LIN {X 0,Y 187.079,Z 92.881,A -85,B 0,C 180,E1 -22258.507,E2 -22258.507} C_VEL
LIN {X 0,Y 185.729,Z 90.066,A -85,B 0,C 180,E1 -22258.924,E2 -22258.924} C_VEL
LIN {X 0,Y 185.6,Z 89.366,A -85,B 0,C 180,E1 -22259.069,E2 -22259.069} C_VEL
LIN {X 0,Y 185.536,Z 89.372,A -85,B 0,C 180,E1 -22263.556,E2 -22263.556} C_VEL
LIN {X 0,Y 185.545,Z 89.369,A -85,B 0,C 180,E1 -22267.304,E2 -22267.304} C_VEL
LIN {X 0,Y 185.487,Z 89.376,A -85,B 0,C 180,E1 -22270.731,E2 -22270.731} C_VEL
LIN {X 0,Y 185.461,Z 89.378,A -85,B 0,C 180,E1 -22276.055,E2 -22276.055} C_VEL
LIN {X 0,Y 185.469,Z 89.375,A -85,B 0,C 180,E1 -22279.896,E2 -22279.896} C_VEL
LIN {X 0,Y 185.508,Z 89.375,A -85,B 0,C 180,E1 -22282.712,E2 -22282.712} C_VEL
LIN {X 0,Y 185.548,Z 89.369,A -85,B 0,C 180,E1 -22287.976,E2 -22287.976} C_VEL
LIN {X 0,Y 185.584,Z 89.362,A -85,B 0,C 180,E1 -22290.576,E2 -22290.576} C_VEL
LIN {X 0,Y 185.59,Z 89.361,A -85,B 0,C 180,E1 -22295.383,E2 -22295.383} C_VEL
LIN {X 0,Y 185.61,Z 89.358,A -85,B 0,C 180,E1 -22300.076,E2 -22300.076} C_VEL
LIN {X 0,Y 185.698,Z 89.324,A -85,B 0,C 180,E1 -22304.638,E2 -22304.638} C_VEL
LIN {X 0,Y 185.891,Z 89.329,A -85,B 0,C 180,E1 -22309.418,E2 -22309.418} C_VEL
LIN {X 0,Y 185.949,Z 89.301,A -85,B 0,C 180,E1 -22313.49,E2 -22313.49} C_VEL
LIN {X 0,Y 186.208,Z 89.273,A -85,B 0,C 180,E1 -22317.837,E2 -22317.837} C_VEL
LIN {X 0,Y 186.41,Z 89.262,A -85,B 0,C 180,E1 -22320,E2 -22320} C_VEL
LIN {X 0,Y 185.915,Z 89.319,A -85,B 0,C 180,E1 -22324.336,E2 -22324.336} C_VEL
LIN {X 0,Y 185.982,Z 89.316,A -85,B 0,C 180,E1 -22328.694,E2 -22328.694} C_VEL
LIN {X 0,Y 185.726,Z 89.351,A -85,B 0,C 180,E1 -22333.123,E2 -22333.123} C_VEL
LIN {X 0,Y 185.689,Z 89.356,A -85,B 0,C 180,E1 -22337.625,E2 -22337.625} C_VEL
LIN {X 0,Y 185.578,Z 89.369,A -85,B 0,C 180,E1 -22342.254,E2 -22342.254} C_VEL
LIN {X 0,Y 185.513,Z 89.381,A -85,B 0,C 180,E1 -22347.04,E2 -22347.04} C_VEL
LIN {X 0,Y 185.546,Z 89.375,A -85,B 0,C 180,E1 -22349.499,E2 -22349.499} C_VEL
LIN {X 0,Y 185.501,Z 89.381,A -85,B 0,C 180,E1 -22354.632,E2 -22354.632} C_VEL
LIN {X 0,Y 185.508,Z 89.378,A -85,B 0,C 180,E1 -22357.313,E2 -22357.313} C_VEL
LIN {X 0,Y 185.474,Z 89.382,A -85,B 0,C 180,E1 -22360.725,E2 -22360.725} C_VEL
LIN {X 0,Y 185.463,Z 89.382,A -85,B 0,C 180,E1 -22366.054,E2 -22366.054} C_VEL
LIN {X 0,Y 185.447,Z 89.388,A -85,B 0,C 180,E1 -22366.815,E2 -22366.815} C_VEL
LIN {X 0,Y 187.546,Z 97.212,A -85,B 0,C 180,E1 -22371.041,E2 -22371.041} C_VEL
LIN {X 0,Y 194.525,Z 112.749,A -85,B 0,C 180,E1 -22373.096,E2 -22373.096} C_VEL
LIN {X 0,Y 199.839,Z 126.939,A -85,B 0,C 180,E1 -22374.634,E2 -22374.634} C_VEL
LIN {X 0,Y 202.047,Z 149.722,A -85,B 0,C 180,E1 -22375.924,E2 -22375.924} C_VEL
LIN {X 0,Y 203.001,Z 161.188,A -85,B 0,C 180,E1 -22376.533,E2 -22376.533} C_VEL
LIN {X 0,Y 201.967,Z 186.96,A -85,B 0,C 180,E1 -22377.398,E2 -22377.398} C_VEL
LIN {X 0,Y 201.164,Z 192.812,A -85,B 0,C 180,E1 -22377.503,E2 -22377.503} C_VEL
LIN {X 0,Y 195.507,Z 209.786,A -85,B 0,C 180,E1 -22377.456,E2 -22377.456} C_VEL
LIN {X 0,Y 194.095,Z 215.48,A -85,B 0,C 180,E1 -22377.666,E2 -22377.666} C_VEL
LIN {X 0,Y 193.836,Z 217.383,A -85,B 0,C 180,E1 -22377.795,E2 -22377.795} C_VEL
LIN {X 0,Y 192.139,Z 229.824,A -85,B 0,C 180,E1 -22378.891,E2 -22378.891} C_VEL
LIN {X 0,Y 189.978,Z 241.772,A -85,B 0,C 180,E1 -22380.344,E2 -22380.344} C_VEL
LIN {X 0,Y 187.729,Z 252.645,A -85,B 0,C 180,E1 -22382.097,E2 -22382.097} C_VEL
LIN {X 0,Y 185.608,Z 261.462,A -85,B 0,C 180,E1 -22383.884,E2 -22383.884} C_VEL
LIN {X 0,Y 183.397,Z 270.914,A -85,B 0,C 180,E1 -22386.273,E2 -22386.273} C_VEL
LIN {X 0,Y 181.019,Z 279.181,A -85,B 0,C 180,E1 -22388.842,E2 -22388.842} C_VEL
LIN {X 0,Y 179.368,Z 286.6,A -85,B 0,C 180,E1 -22391.732,E2 -22391.732} C_VEL
LIN {X 0,Y 177.815,Z 293.562,A -85,B 0,C 180,E1 -22395.113,E2 -22395.113} C_VEL
LIN {X 0,Y 176.781,Z 299.125,A -85,B 0,C 180,E1 -22398.534,E2 -22398.534} C_VEL
LIN {X 0,Y 176.302,Z 303.475,A -85,B 0,C 180,E1 -22401.98,E2 -22401.98} C_VEL
LIN {X 0,Y 176.263,Z 306.729,A -85,B 0,C 180,E1 -22405.426,E2 -22405.426} C_VEL
LIN {X 0,Y 176.338,Z 308.334,A -85,B 0,C 180,E1 -22407.716,E2 -22407.716} C_VEL
LIN {X 0,Y 176.495,Z 309.519,A -85,B 0,C 180,E1 -22410,E2 -22410} C_VEL
LIN {X 0,Y 176.316,Z 310.226,A -85,B 0,C 180,E1 -22412.284,E2 -22412.284} C_VEL
LIN {X 0,Y 176.232,Z 310.534,A -85,B 0,C 180,E1 -22414.575,E2 -22414.575} C_VEL
LIN {X 0,Y 176.383,Z 309.99,A -85,B 0,C 180,E1 -22419.171,E2 -22419.171} C_VEL
LIN {X 0,Y 176.861,Z 309.117,A -85,B 0,C 180,E1 -22421.46,E2 -22421.46} C_VEL
LIN {X 0,Y 178.546,Z 306.157,A -85,B 0,C 180,E1 -22425.994,E2 -22425.994} C_VEL
LIN {X 0,Y 180.7,Z 302.835,A -85,B 0,C 180,E1 -22429.305,E2 -22429.305} C_VEL
LIN {X 0,Y 183.398,Z 298.468,A -85,B 0,C 180,E1 -22432.533,E2 -22432.533} C_VEL
LIN {X 0,Y 187.098,Z 291.917,A -85,B 0,C 180,E1 -22436.191,E2 -22436.191} C_VEL
LIN {X 0,Y 191.062,Z 284.767,A -85,B 0,C 180,E1 -22439.169,E2 -22439.169} C_VEL
LIN {X 0,Y 195.634,Z 275.903,A -85,B 0,C 180,E1 -22441.998,E2 -22441.998} C_VEL
LIN {X 0,Y 200.264,Z 265.844,A -85,B 0,C 180,E1 -22444.464,E2 -22444.464} C_VEL
LIN {X 0,Y 204.349,Z 255.58,A -85,B 0,C 180,E1 -22446.389,E2 -22446.389} C_VEL
LIN {X 0,Y 208.228,Z 244.222,A -85,B 0,C 180,E1 -22448.022,E2 -22448.022} C_VEL
LIN {X 0,Y 211.569,Z 232.42,A -85,B 0,C 180,E1 -22449.289,E2 -22449.289} C_VEL
LIN {X 0,Y 214.263,Z 219.437,A -85,B 0,C 180,E1 -22450.3,E2 -22450.3} C_VEL
LIN {X 0,Y 216.25,Z 205.853,A -85,B 0,C 180,E1 -22450.98,E2 -22450.98} C_VEL
LIN {X 0,Y 218.563,Z 169.214,A -85,B 0,C 180,E1 -22452.133,E2 -22452.133} C_VEL
LIN {X 0,Y 217.377,Z 159.103,A -85,B 0,C 180,E1 -22452.939,E2 -22452.939} C_VEL
LIN {X 0,Y 211.594,Z 145.25,A -85,B 0,C 180,E1 -22455.352,E2 -22455.352} C_VEL
LIN {X 0,Y 206.029,Z 134.045,A -85,B 0,C 180,E1 -22457.813,E2 -22457.813} C_VEL
LIN {X 0,Y 201.532,Z 125.851,A -85,B 0,C 180,E1 -22459.965,E2 -22459.965} C_VEL
LIN {X 0,Y 196.559,Z 117.494,A -85,B 0,C 180,E1 -22462.566,E2 -22462.566} C_VEL
LIN {X 0,Y 192.905,Z 111.765,A -85,B 0,C 180,E1 -22464.664,E2 -22464.664} C_VEL
LIN {X 0,Y 188.825,Z 105.716,A -85,B 0,C 180,E1 -22467.254,E2 -22467.254} C_VEL
LIN {X 0,Y 185.057,Z 100.378,A -85,B 0,C 180,E1 -22469.954,E2 -22469.954} C_VEL
LIN {X 0,Y 183.131,Z 97.941,A -85,B 0,C 180,E1 -22471.462,E2 -22471.462} C_VEL
LIN {X 0,Y 180.355,Z 94.307,A -85,B 0,C 180,E1 -22473.883,E2 -22473.883} C_VEL
LIN {X 0,Y 179.145,Z 92.283,A -85,B 0,C 180,E1 -22475.199,E2 -22475.199} C_VEL
LIN {X 0,Y 178.547,Z 90.23,A -85,B 0,C 180,E1 -22478.041,E2 -22478.041} C_VEL
LIN {X 0,Y 178.673,Z 90.218,A -85,B 0,C 180,E1 -22481.658,E2 -22481.658} C_VEL
LIN {X 0,Y 178.661,Z 90.221,A -85,B 0,C 180,E1 -22486.348,E2 -22486.348} C_VEL
LIN {X 0,Y 178.914,Z 90.196,A -85,B 0,C 180,E1 -22490.96,E2 -22490.96} C_VEL
LIN {X 0,Y 179.154,Z 90.152,A -85,B 0,C 180,E1 -22497.752,E2 -22497.752} C_VEL
LIN {X 0,Y 179.372,Z 90.132,A -85,B 0,C 180,E1 -22500,E2 -22500} C_VEL
LIN {X 0,Y 178.866,Z 90.189,A -85,B 0,C 180,E1 -22504.507,E2 -22504.507} C_VEL
LIN {X 0,Y 178.912,Z 90.181,A -85,B 0,C 180,E1 -22509.04,E2 -22509.04} C_VEL
LIN {X 0,Y 178.652,Z 90.367,A -85,B 0,C 180,E1 -22515.034,E2 -22515.034} C_VEL
LIN {X 0,Y 179.507,Z 92.842,A -85,B 0,C 180,E1 -22516.052,E2 -22516.052} C_VEL
LIN {X 0,Y 181.383,Z 94.994,A -85,B 0,C 180,E1 -22517.766,E2 -22517.766} C_VEL
LIN {X 0,Y 183.423,Z 96.333,A -85,B 0,C 180,E1 -22519.371,E2 -22519.371} C_VEL
LIN {X 0,Y 185.032,Z 99.289,A -85,B 0,C 180,E1 -22520.714,E2 -22520.714} C_VEL
LIN {X 0,Y 187.677,Z 101.543,A -85,B 0,C 180,E1 -22522.533,E2 -22522.533} C_VEL
LIN {X 0,Y 190.252,Z 105.409,A -85,B 0,C 180,E1 -22524.286,E2 -22524.286} C_VEL
LIN {X 0,Y 192.095,Z 107.229,A -85,B 0,C 180,E1 -22525.388,E2 -22525.388} C_VEL
LIN {X 0,Y 194.769,Z 110.861,A -85,B 0,C 180,E1 -22526.956,E2 -22526.956} C_VEL
LIN {X 0,Y 196.441,Z 113.104,A -85,B 0,C 180,E1 -22527.876,E2 -22527.876} C_VEL
LIN {X 0,Y 199.512,Z 117.279,A -85,B 0,C 180,E1 -22529.476,E2 -22529.476} C_VEL
LIN {X 0,Y 204.379,Z 124.152,A -85,B 0,C 180,E1 -22531.81,E2 -22531.81} C_VEL
LIN {X 0,Y 211.211,Z 134.963,A -85,B 0,C 180,E1 -22534.777,E2 -22534.777} C_VEL
LIN {X 0,Y 217.553,Z 146.272,A -85,B 0,C 180,E1 -22537.28,E2 -22537.28} C_VEL
LIN {X 0,Y 219.698,Z 150.374,A -85,B 0,C 180,E1 -22538.082,E2 -22538.082} C_VEL
LIN {X 0,Y 217.14,Z 189.325,A -85,B 0,C 180,E1 -22539.281,E2 -22539.281} C_VEL
LIN {X 0,Y 215.488,Z 202.678,A -85,B 0,C 180,E1 -22540.031,E2 -22540.031} C_VEL
LIN {X 0,Y 213.455,Z 214.164,A -85,B 0,C 180,E1 -22540.995,E2 -22540.995} C_VEL
LIN {X 0,Y 210.553,Z 226.047,A -85,B 0,C 180,E1 -22542.313,E2 -22542.313} C_VEL
LIN {X 0,Y 207.233,Z 236.837,A -85,B 0,C 180,E1 -22543.89,E2 -22543.89} C_VEL
LIN {X 0,Y 203.257,Z 247.568,A -85,B 0,C 180,E1 -22545.904,E2 -22545.904} C_VEL
LIN {X 0,Y 199.599,Z 256.292,A -85,B 0,C 180,E1 -22548.01,E2 -22548.01} C_VEL
LIN {X 0,Y 195.695,Z 264.272,A -85,B 0,C 180,E1 -22550.397,E2 -22550.397} C_VEL
LIN {X 0,Y 191.556,Z 272,A -85,B 0,C 180,E1 -22553.402,E2 -22553.402} C_VEL
LIN {X 0,Y 187.26,Z 279.067,A -85,B 0,C 180,E1 -22557.03,E2 -22557.03} C_VEL
LIN {X 0,Y 184.152,Z 283.709,A -85,B 0,C 180,E1 -22560.255,E2 -22560.255} C_VEL
LIN {X 0,Y 182.382,Z 286.142,A -85,B 0,C 180,E1 -22562.457,E2 -22562.457} C_VEL
LIN {X 0,Y 180.863,Z 288.109,A -85,B 0,C 180,E1 -22564.695,E2 -22564.695} C_VEL
LIN {X 0,Y 179.569,Z 289.65,A -85,B 0,C 180,E1 -22566.959,E2 -22566.959} C_VEL
LIN {X 0,Y 178.48,Z 290.741,A -85,B 0,C 180,E1 -22569.244,E2 -22569.244} C_VEL
LIN {X 0,Y 177.61,Z 291.439,A -85,B 0,C 180,E1 -22571.746,E2 -22571.746} C_VEL
LIN {X 0,Y 176.514,Z 291.56,A -85,B 0,C 180,E1 -22576.179,E2 -22576.179} C_VEL
LIN {X 0,Y 176.263,Z 291.008,A -85,B 0,C 180,E1 -22578.5,E2 -22578.5} C_VEL
LIN {X 0,Y 176.402,Z 288.697,A -85,B 0,C 180,E1 -22583.136,E2 -22583.136} C_VEL
LIN {X 0,Y 176.854,Z 285.866,A -85,B 0,C 180,E1 -22586.583,E2 -22586.583} C_VEL
LIN {X 0,Y 177.509,Z 282.036,A -85,B 0,C 180,E1 -22590,E2 -22590} C_VEL
LIN {X 0,Y 178.57,Z 277.089,A -85,B 0,C 180,E1 -22593.385,E2 -22593.385} C_VEL
LIN {X 0,Y 180.129,Z 270.873,A -85,B 0,C 180,E1 -22596.722,E2 -22596.722} C_VEL
LIN {X 0,Y 182.228,Z 263.095,A -85,B 0,C 180,E1 -22599.995,E2 -22599.995} C_VEL
LIN {X 0,Y 184.684,Z 253.401,A -85,B 0,C 180,E1 -22603.199,E2 -22603.199} C_VEL
LIN {X 0,Y 187.279,Z 243.315,A -85,B 0,C 180,E1 -22605.788,E2 -22605.788} C_VEL
LIN {X 0,Y 189.62,Z 233.3,A -85,B 0,C 180,E1 -22607.805,E2 -22607.805} C_VEL
LIN {X 0,Y 191.652,Z 222.453,A -85,B 0,C 180,E1 -22609.55,E2 -22609.55} C_VEL
LIN {X 0,Y 193.437,Z 210.502,A -85,B 0,C 180,E1 -22611.026,E2 -22611.026} C_VEL
LIN {X 0,Y 194.843,Z 197.397,A -85,B 0,C 180,E1 -22612.186,E2 -22612.186} C_VEL
LIN {X 0,Y 195.736,Z 184.28,A -85,B 0,C 180,E1 -22612.914,E2 -22612.914} C_VEL
LIN {X 0,Y 198.224,Z 129.371,A -85,B 0,C 180,E1 -22614.791,E2 -22614.791} C_VEL
LIN {X 0,Y 194.633,Z 120.748,A -85,B 0,C 180,E1 -22615.793,E2 -22615.793} C_VEL
LIN {X 0,Y 187.561,Z 106.659,A -85,B 0,C 180,E1 -22617.78,E2 -22617.78} C_VEL
LIN {X 0,Y 181.804,Z 96.696,A -85,B 0,C 180,E1 -22619.473,E2 -22619.473} C_VEL
LIN {X 0,Y 180.363,Z 94.19,A -85,B 0,C 180,E1 -22619.92,E2 -22619.92} C_VEL
LIN {X 0,Y 178.803,Z 91.62,A -85,B 0,C 180,E1 -22620.409,E2 -22620.409} C_VEL
LIN {X 0,Y 178.493,Z 90.248,A -85,B 0,C 180,E1 -22620.599,E2 -22620.599} C_VEL
LIN {X 0,Y 178.496,Z 90.248,A -85,B 0,C 180,E1 -22624.225,E2 -22624.225} C_VEL
LIN {X 0,Y 178.42,Z 90.26,A -85,B 0,C 180,E1 -22629.069,E2 -22629.069} C_VEL
LIN {X 0,Y 178.405,Z 90.258,A -85,B 0,C 180,E1 -22632.044,E2 -22632.044} C_VEL
LIN {X 0,Y 178.395,Z 90.256,A -85,B 0,C 180,E1 -22635.164,E2 -22635.164} C_VEL
LIN {X 0,Y 178.404,Z 90.259,A -85,B 0,C 180,E1 -22638.46,E2 -22638.46} C_VEL
LIN {X 0,Y 178.425,Z 90.252,A -85,B 0,C 180,E1 -22643.784,E2 -22643.784} C_VEL
LIN {X 0,Y 178.489,Z 90.249,A -85,B 0,C 180,E1 -22646.547,E2 -22646.547} C_VEL
LIN {X 0,Y 178.525,Z 90.24,A -85,B 0,C 180,E1 -22650.007,E2 -22650.007} C_VEL
LIN {X 0,Y 178.537,Z 90.239,A -85,B 0,C 180,E1 -22654.876,E2 -22654.876} C_VEL
LIN {X 0,Y 178.626,Z 90.222,A -85,B 0,C 180,E1 -22660.784,E2 -22660.784} C_VEL
LIN {X 0,Y 178.662,Z 90.215,A -85,B 0,C 180,E1 -22666.348,E2 -22666.348} C_VEL
LIN {X 0,Y 178.914,Z 90.195,A -85,B 0,C 180,E1 -22670.96,E2 -22670.96} C_VEL
LIN {X 0,Y 179.154,Z 90.15,A -85,B 0,C 180,E1 -22677.752,E2 -22677.752} C_VEL
LIN {X 0,Y 179.373,Z 90.138,A -85,B 0,C 180,E1 -22680,E2 -22680} C_VEL
LIN {X 0,Y 178.862,Z 90.197,A -85,B 0,C 180,E1 -22684.508,E2 -22684.508} C_VEL
LIN {X 0,Y 178.911,Z 90.195,A -85,B 0,C 180,E1 -22689.041,E2 -22689.041} C_VEL
LIN {X 0,Y 178.655,Z 90.23,A -85,B 0,C 180,E1 -22693.653,E2 -22693.653} C_VEL
LIN {X 0,Y 178.624,Z 90.233,A -85,B 0,C 180,E1 -22699.214,E2 -22699.214} C_VEL
LIN {X 0,Y 178.518,Z 90.245,A -85,B 0,C 180,E1 -22705.111,E2 -22705.111} C_VEL
LIN {X 0,Y 178.463,Z 90.258,A -85,B 0,C 180,E1 -22710.794,E2 -22710.794} C_VEL
LIN {X 0,Y 178.486,Z 90.254,A -85,B 0,C 180,E1 -22714.218,E2 -22714.218} C_VEL
LIN {X 0,Y 178.398,Z 90.263,A -85,B 0,C 180,E1 -22719.074,E2 -22719.074} C_VEL
LIN {X 0,Y 178.401,Z 90.263,A -85,B 0,C 180,E1 -22722.045,E2 -22722.045} C_VEL
LIN {X 0,Y 178.418,Z 90.378,A -85,B 0,C 180,E1 -22725.76,E2 -22725.76} C_VEL
LIN {X 0,Y 180.164,Z 96.881,A -85,B 0,C 180,E1 -22729.415,E2 -22729.415} C_VEL
LIN {X 0,Y 186.535,Z 110.257,A -85,B 0,C 180,E1 -22731.427,E2 -22731.427} C_VEL
LIN {X 0,Y 192.601,Z 125.371,A -85,B 0,C 180,E1 -22733.283,E2 -22733.283} C_VEL
LIN {X 0,Y 193.865,Z 128.929,A -85,B 0,C 180,E1 -22733.668,E2 -22733.668} C_VEL
LIN {X 0,Y 195.93,Z 151.227,A -85,B 0,C 180,E1 -22734.975,E2 -22734.975} C_VEL
LIN {X 0,Y 196.76,Z 162.292,A -85,B 0,C 180,E1 -22735.576,E2 -22735.576} C_VEL
LIN {X 0,Y 194.789,Z 206.829,A -85,B 0,C 180,E1 -22737.161,E2 -22737.161} C_VEL
LIN {X 0,Y 193.836,Z 217.383,A -85,B 0,C 180,E1 -22737.795,E2 -22737.795} C_VEL
LIN {X 0,Y 193.089,Z 221.163,A -85,B 0,C 180,E1 -22738.044,E2 -22738.044} C_VEL
LIN {X 0,Y 190.241,Z 228.451,A -85,B 0,C 180,E1 -22738.439,E2 -22738.439} C_VEL
LIN {X 0,Y 184.998,Z 238.939,A -85,B 0,C 180,E1 -22739.182,E2 -22739.182} C_VEL
LIN {X 0,Y 183.098,Z 244.152,A -85,B 0,C 180,E1 -22739.822,E2 -22739.822} C_VEL
LIN {X 0,Y 182.711,Z 245.852,A -85,B 0,C 180,E1 -22740.091,E2 -22740.091} C_VEL
LIN {X 0,Y 180.095,Z 256.718,A -85,B 0,C 180,E1 -22742.076,E2 -22742.076} C_VEL
LIN {X 0,Y 177.533,Z 266.947,A -85,B 0,C 180,E1 -22744.5,E2 -22744.5} C_VEL
LIN {X 0,Y 175.322,Z 275.52,A -85,B 0,C 180,E1 -22747.058,E2 -22747.058} C_VEL
LIN {X 0,Y 173.589,Z 281.649,A -85,B 0,C 180,E1 -22749.252,E2 -22749.252} C_VEL
LIN {X 0,Y 171.721,Z 289.545,A -85,B 0,C 180,E1 -22752.739,E2 -22752.739} C_VEL
LIN {X 0,Y 170.071,Z 296.759,A -85,B 0,C 180,E1 -22756.863,E2 -22756.863} C_VEL
LIN {X 0,Y 169.361,Z 301.565,A -85,B 0,C 180,E1 -22760.445,E2 -22760.445} C_VEL
LIN {X 0,Y 169.124,Z 305.224,A -85,B 0,C 180,E1 -22764.037,E2 -22764.037} C_VEL
LIN {X 0,Y 169.255,Z 307.84,A -85,B 0,C 180,E1 -22767.62,E2 -22767.62} C_VEL
LIN {X 0,Y 169.429,Z 309.056,A -85,B 0,C 180,E1 -22770,E2 -22770} C_VEL
LIN {X 0,Y 169.153,Z 310.116,A -85,B 0,C 180,E1 -22774.316,E2 -22774.316} C_VEL
LIN {X 0,Y 169.086,Z 310.075,A -85,B 0,C 180,E1 -22777.163,E2 -22777.163} C_VEL
LIN {X 0,Y 169.857,Z 308.813,A -85,B 0,C 180,E1 -22781.939,E2 -22781.939} C_VEL
LIN {X 0,Y 171.721,Z 305.907,A -85,B 0,C 180,E1 -22786.648,E2 -22786.648} C_VEL
LIN {X 0,Y 173.969,Z 302.637,A -85,B 0,C 180,E1 -22790.083,E2 -22790.083} C_VEL
LIN {X 0,Y 176.824,Z 298.327,A -85,B 0,C 180,E1 -22793.419,E2 -22793.419} C_VEL
LIN {X 0,Y 180.722,Z 291.842,A -85,B 0,C 180,E1 -22797.19,E2 -22797.19} C_VEL
LIN {X 0,Y 184.879,Z 284.794,A -85,B 0,C 180,E1 -22800.244,E2 -22800.244} C_VEL
LIN {X 0,Y 189.648,Z 276.013,A -85,B 0,C 180,E1 -22803.135,E2 -22803.135} C_VEL
LIN {X 0,Y 194.47,Z 266.071,A -85,B 0,C 180,E1 -22805.644,E2 -22805.644} C_VEL
LIN {X 0,Y 198.691,Z 255.981,A -85,B 0,C 180,E1 -22807.601,E2 -22807.601} C_VEL
LIN {X 0,Y 202.702,Z 244.802,A -85,B 0,C 180,E1 -22809.254,E2 -22809.254} C_VEL
LIN {X 0,Y 206.425,Z 232.262,A -85,B 0,C 180,E1 -22810.627,E2 -22810.627} C_VEL
LIN {X 0,Y 209.214,Z 219.401,A -85,B 0,C 180,E1 -22811.644,E2 -22811.644} C_VEL
LIN {X 0,Y 211.219,Z 206.356,A -85,B 0,C 180,E1 -22812.311,E2 -22812.311} C_VEL
LIN {X 0,Y 213.641,Z 170.417,A -85,B 0,C 180,E1 -22813.466,E2 -22813.466} C_VEL
LIN {X 0,Y 212.726,Z 162.146,A -85,B 0,C 180,E1 -22814.147,E2 -22814.147} C_VEL
LIN {X 0,Y 207.357,Z 149.125,A -85,B 0,C 180,E1 -22816.53,E2 -22816.53} C_VEL
LIN {X 0,Y 202.042,Z 138.081,A -85,B 0,C 180,E1 -22819.045,E2 -22819.045} C_VEL
LIN {X 0,Y 196.613,Z 128.146,A -85,B 0,C 180,E1 -22821.85,E2 -22821.85} C_VEL
LIN {X 0,Y 193.113,Z 122.307,A -85,B 0,C 180,E1 -22823.825,E2 -22823.825} C_VEL
LIN {X 0,Y 190.334,Z 117.733,A -85,B 0,C 180,E1 -22825.529,E2 -22825.529} C_VEL
LIN {X 0,Y 186.434,Z 111.75,A -85,B 0,C 180,E1 -22828.146,E2 -22828.146} C_VEL
LIN {X 0,Y 182.795,Z 106.363,A -85,B 0,C 180,E1 -22830.911,E2 -22830.911} C_VEL
LIN {X 0,Y 177.729,Z 99.455,A -85,B 0,C 180,E1 -22835.51,E2 -22835.51} C_VEL
LIN {X 0,Y 175.025,Z 96.393,A -85,B 0,C 180,E1 -22838.505,E2 -22838.505} C_VEL
LIN {X 0,Y 172.883,Z 94.324,A -85,B 0,C 180,E1 -22841.329,E2 -22841.329} C_VEL
LIN {X 0,Y 171.786,Z 92.097,A -85,B 0,C 180,E1 -22843.282,E2 -22843.282} C_VEL
LIN {X 0,Y 171.586,Z 91.097,A -85,B 0,C 180,E1 -22843.873,E2 -22843.873} C_VEL
LIN {X 0,Y 171.85,Z 91.08,A -85,B 0,C 180,E1 -22850.585,E2 -22850.585} C_VEL
LIN {X 0,Y 171.818,Z 91.08,A -85,B 0,C 180,E1 -22855.307,E2 -22855.307} C_VEL
LIN {X 0,Y 172.335,Z 91.008,A -85,B 0,C 180,E1 -22860,E2 -22860} C_VEL
LIN {X 0,Y 171.814,Z 91.068,A -85,B 0,C 180,E1 -22864.692,E2 -22864.692} C_VEL
LIN {X 0,Y 171.885,Z 91.271,A -85,B 0,C 180,E1 -22867.488,E2 -22867.488} C_VEL
LIN {X 0,Y 172.525,Z 93.251,A -85,B 0,C 180,E1 -22868.787,E2 -22868.787} C_VEL
LIN {X 0,Y 174.365,Z 95.792,A -85,B 0,C 180,E1 -22871.475,E2 -22871.475} C_VEL
LIN {X 0,Y 176.872,Z 97.237,A -85,B 0,C 180,E1 -22874.232,E2 -22874.232} C_VEL
LIN {X 0,Y 178.186,Z 100.016,A -85,B 0,C 180,E1 -22875.733,E2 -22875.733} C_VEL
LIN {X 0,Y 180.534,Z 102.228,A -85,B 0,C 180,E1 -22877.852,E2 -22877.852} C_VEL
LIN {X 0,Y 181.461,Z 102.963,A -85,B 0,C 180,E1 -22878.611,E2 -22878.611} C_VEL
LIN {X 0,Y 183.559,Z 106.305,A -85,B 0,C 180,E1 -22880.376,E2 -22880.376} C_VEL
LIN {X 0,Y 185.749,Z 108.325,A -85,B 0,C 180,E1 -22881.939,E2 -22881.939} C_VEL
LIN {X 0,Y 188.215,Z 111.879,A -85,B 0,C 180,E1 -22883.666,E2 -22883.666} C_VEL
LIN {X 0,Y 189.886,Z 113.752,A -85,B 0,C 180,E1 -22884.72,E2 -22884.72} C_VEL
LIN {X 0,Y 193.951,Z 119.332,A -85,B 0,C 180,E1 -22887.151,E2 -22887.151} C_VEL
LIN {X 0,Y 197.722,Z 124.622,A -85,B 0,C 180,E1 -22889.185,E2 -22889.185} C_VEL
LIN {X 0,Y 202.306,Z 131.456,A -85,B 0,C 180,E1 -22891.451,E2 -22891.451} C_VEL
LIN {X 0,Y 208.135,Z 140.952,A -85,B 0,C 180,E1 -22894.077,E2 -22894.077} C_VEL
LIN {X 0,Y 214.692,Z 153.106,A -85,B 0,C 180,E1 -22896.776,E2 -22896.776} C_VEL
LIN {X 0,Y 212.202,Z 189.729,A -85,B 0,C 180,E1 -22897.925,E2 -22897.925} C_VEL
LIN {X 0,Y 210.489,Z 203.084,A -85,B 0,C 180,E1 -22898.685,E2 -22898.685} C_VEL
LIN {X 0,Y 208.186,Z 215.487,A -85,B 0,C 180,E1 -22899.749,E2 -22899.749} C_VEL
LIN {X 0,Y 205.125,Z 227.154,A -85,B 0,C 180,E1 -22901.082,E2 -22901.082} C_VEL
LIN {X 0,Y 201.318,Z 238.818,A -85,B 0,C 180,E1 -22902.852,E2 -22902.852} C_VEL
LIN {X 0,Y 197.645,Z 248.181,A -85,B 0,C 180,E1 -22904.669,E2 -22904.669} C_VEL
LIN {X 0,Y 193.421,Z 257.736,A -85,B 0,C 180,E1 -22907.056,E2 -22907.056} C_VEL
LIN {X 0,Y 188.602,Z 266.875,A -85,B 0,C 180,E1 -22909.999,E2 -22909.999} C_VEL
LIN {X 0,Y 184.186,Z 274.505,A -85,B 0,C 180,E1 -22913.254,E2 -22913.254} C_VEL
LIN {X 0,Y 180.008,Z 280.796,A -85,B 0,C 180,E1 -22916.866,E2 -22916.866} C_VEL
LIN {X 0,Y 176.893,Z 285.113,A -85,B 0,C 180,E1 -22920.223,E2 -22920.223} C_VEL
LIN {X 0,Y 174.312,Z 288.321,A -85,B 0,C 180,E1 -22923.672,E2 -22923.672} C_VEL
LIN {X 0,Y 172.887,Z 289.896,A -85,B 0,C 180,E1 -22926.014,E2 -22926.014} C_VEL
LIN {X 0,Y 171.728,Z 291.048,A -85,B 0,C 180,E1 -22928.388,E2 -22928.388} C_VEL
LIN {X 0,Y 170.593,Z 291.854,A -85,B 0,C 180,E1 -22931.359,E2 -22931.359} C_VEL
LIN {X 0,Y 169.531,Z 291.966,A -85,B 0,C 180,E1 -22935.598,E2 -22935.598} C_VEL
LIN {X 0,Y 169.214,Z 291.477,A -85,B 0,C 180,E1 -22938.015,E2 -22938.015} C_VEL
LIN {X 0,Y 169.268,Z 289.231,A -85,B 0,C 180,E1 -22942.845,E2 -22942.845} C_VEL
LIN {X 0,Y 169.739,Z 286.463,A -85,B 0,C 180,E1 -22946.439,E2 -22946.439} C_VEL
LIN {X 0,Y 170.381,Z 282.704,A -85,B 0,C 180,E1 -22950,E2 -22950} C_VEL
LIN {X 0,Y 171.506,Z 277.829,A -85,B 0,C 180,E1 -22953.524,E2 -22953.524} C_VEL
LIN {X 0,Y 173.096,Z 271.697,A -85,B 0,C 180,E1 -22956.997,E2 -22956.997} C_VEL
LIN {X 0,Y 175.284,Z 264.059,A -85,B 0,C 180,E1 -22960.395,E2 -22960.395} C_VEL
LIN {X 0,Y 177.813,Z 254.485,A -85,B 0,C 180,E1 -22963.719,E2 -22963.719} C_VEL
LIN {X 0,Y 180.472,Z 244.58,A -85,B 0,C 180,E1 -22966.4,E2 -22966.4} C_VEL
LIN {X 0,Y 182.918,Z 234.796,A -85,B 0,C 180,E1 -22968.481,E2 -22968.481} C_VEL
LIN {X 0,Y 185.049,Z 224.218,A -85,B 0,C 180,E1 -22970.277,E2 -22970.277} C_VEL
LIN {X 0,Y 187.057,Z 211.535,A -85,B 0,C 180,E1 -22971.924,E2 -22971.924} C_VEL
LIN {X 0,Y 188.529,Z 198.803,A -85,B 0,C 180,E1 -22973.116,E2 -22973.116} C_VEL
LIN {X 0,Y 189.452,Z 186.403,A -85,B 0,C 180,E1 -22973.865,E2 -22973.865} C_VEL
LIN {X 0,Y 192.002,Z 130.643,A -85,B 0,C 180,E1 -22975.851,E2 -22975.851} C_VEL
LIN {X 0,Y 185.329,Z 116.24,A -85,B 0,C 180,E1 -22977.801,E2 -22977.801} C_VEL
LIN {X 0,Y 178.679,Z 103.908,A -85,B 0,C 180,E1 -22979.836,E2 -22979.836} C_VEL
LIN {X 0,Y 174.98,Z 97.881,A -85,B 0,C 180,E1 -22981.018,E2 -22981.018} C_VEL
LIN {X 0,Y 173.262,Z 95.093,A -85,B 0,C 180,E1 -22981.59,E2 -22981.59} C_VEL
LIN {X 0,Y 171.822,Z 92.792,A -85,B 0,C 180,E1 -22982.08,E2 -22982.08} C_VEL
LIN {X 0,Y 171.394,Z 91.137,A -85,B 0,C 180,E1 -22982.296,E2 -22982.296} C_VEL
LIN {X 0,Y 171.407,Z 91.133,A -85,B 0,C 180,E1 -22985.032,E2 -22985.032} C_VEL
LIN {X 0,Y 171.381,Z 91.136,A -85,B 0,C 180,E1 -22988.817,E2 -22988.817} C_VEL
LIN {X 0,Y 171.323,Z 91.14,A -85,B 0,C 180,E1 -22994.217,E2 -22994.217} C_VEL
LIN {X 0,Y 171.336,Z 91.136,A -85,B 0,C 180,E1 -22998.982,E2 -22998.982} C_VEL
LIN {X 0,Y 171.389,Z 91.134,A -85,B 0,C 180,E1 -23002.042,E2 -23002.042} C_VEL
LIN {X 0,Y 171.4,Z 91.127,A -85,B 0,C 180,E1 -23005.093,E2 -23005.093} C_VEL
LIN {X 0,Y 171.452,Z 91.122,A -85,B 0,C 180,E1 -23010.535,E2 -23010.535} C_VEL
LIN {X 0,Y 171.461,Z 91.121,A -85,B 0,C 180,E1 -23015.802,E2 -23015.802} C_VEL
LIN {X 0,Y 171.582,Z 91.098,A -85,B 0,C 180,E1 -23020.872,E2 -23020.872} C_VEL
LIN {X 0,Y 171.579,Z 91.091,A -85,B 0,C 180,E1 -23025.773,E2 -23025.773} C_VEL
LIN {X 0,Y 171.851,Z 91.076,A -85,B 0,C 180,E1 -23030.585,E2 -23030.585} C_VEL
LIN {X 0,Y 171.814,Z 91.047,A -85,B 0,C 180,E1 -23035.308,E2 -23035.308} C_VEL
LIN {X 0,Y 172.336,Z 91.015,A -85,B 0,C 180,E1 -23040,E2 -23040} C_VEL
LIN {X 0,Y 171.811,Z 91.075,A -85,B 0,C 180,E1 -23044.693,E2 -23044.693} C_VEL
LIN {X 0,Y 171.849,Z 91.072,A -85,B 0,C 180,E1 -23049.415,E2 -23049.415} C_VEL
LIN {X 0,Y 171.572,Z 91.111,A -85,B 0,C 180,E1 -23054.228,E2 -23054.228} C_VEL
LIN {X 0,Y 171.543,Z 91.113,A -85,B 0,C 180,E1 -23059.558,E2 -23059.558} C_VEL
LIN {X 0,Y 171.447,Z 91.127,A -85,B 0,C 180,E1 -23065.599,E2 -23065.599} C_VEL
LIN {X 0,Y 171.42,Z 91.135,A -85,B 0,C 180,E1 -23070.573,E2 -23070.573} C_VEL
LIN {X 0,Y 171.395,Z 91.138,A -85,B 0,C 180,E1 -23075.035,E2 -23075.035} C_VEL
LIN {X 0,Y 171.36,Z 91.141,A -85,B 0,C 180,E1 -23078.808,E2 -23078.808} C_VEL
LIN {X 0,Y 171.367,Z 91.284,A -85,B 0,C 180,E1 -23084.552,E2 -23084.552} C_VEL
LIN {X 0,Y 172.713,Z 96.273,A -85,B 0,C 180,E1 -23087.579,E2 -23087.579} C_VEL
LIN {X 0,Y 174.962,Z 100.629,A -85,B 0,C 180,E1 -23088.365,E2 -23088.365} C_VEL
LIN {X 0,Y 180.087,Z 111.356,A -85,B 0,C 180,E1 -23090.095,E2 -23090.095} C_VEL
LIN {X 0,Y 184.61,Z 122.124,A -85,B 0,C 180,E1 -23091.573,E2 -23091.573} C_VEL
LIN {X 0,Y 187.983,Z 131.446,A -85,B 0,C 180,E1 -23092.672,E2 -23092.672} C_VEL
LIN {X 0,Y 190.642,Z 161.189,A -85,B 0,C 180,E1 -23094.474,E2 -23094.474} C_VEL
LIN {X 0,Y 188.658,Z 205.888,A -85,B 0,C 180,E1 -23096.108,E2 -23096.108} C_VEL
LIN {X 0,Y 187.324,Z 219.248,A -85,B 0,C 180,E1 -23096.962,E2 -23096.962} C_VEL
LIN {X 0,Y 185.495,Z 231.462,A -85,B 0,C 180,E1 -23098.125,E2 -23098.125} C_VEL
LIN {X 0,Y 183.146,Z 243.777,A -85,B 0,C 180,E1 -23099.757,E2 -23099.757} C_VEL
LIN {X 0,Y 182.711,Z 245.852,A -85,B 0,C 180,E1 -23100.091,E2 -23100.091} C_VEL
LIN {X 0,Y 181.391,Z 249.288,A -85,B 0,C 180,E1 -23100.586,E2 -23100.586} C_VEL
LIN {X 0,Y 177.453,Z 254.474,A -85,B 0,C 180,E1 -23101.19,E2 -23101.19} C_VEL
LIN {X 0,Y 173.45,Z 259.47,A -85,B 0,C 180,E1 -23101.917,E2 -23101.917} C_VEL
LIN {X 0,Y 172.05,Z 262.576,A -85,B 0,C 180,E1 -23102.601,E2 -23102.601} C_VEL
LIN {X 0,Y 169.87,Z 270.865,A -85,B 0,C 180,E1 -23104.908,E2 -23104.908} C_VEL
LIN {X 0,Y 167.246,Z 279.285,A -85,B 0,C 180,E1 -23107.778,E2 -23107.778} C_VEL
LIN {X 0,Y 165.479,Z 286.319,A -85,B 0,C 180,E1 -23110.783,E2 -23110.783} C_VEL
LIN {X 0,Y 163.791,Z 293.195,A -85,B 0,C 180,E1 -23114.444,E2 -23114.444} C_VEL
LIN {X 0,Y 162.511,Z 299.495,A -85,B 0,C 180,E1 -23118.778,E2 -23118.778} C_VEL
LIN {X 0,Y 162.082,Z 303.581,A -85,B 0,C 180,E1 -23122.525,E2 -23122.525} C_VEL
LIN {X 0,Y 162.103,Z 306.169,A -85,B 0,C 180,E1 -23125.691,E2 -23125.691} C_VEL
LIN {X 0,Y 162.34,Z 308.586,A -85,B 0,C 180,E1 -23130,E2 -23130} C_VEL
LIN {X 0,Y 162.079,Z 309.676,A -85,B 0,C 180,E1 -23134.195,E2 -23134.195} C_VEL
LIN {X 0,Y 162.01,Z 309.7,A -85,B 0,C 180,E1 -23137.478,E2 -23137.478} C_VEL
LIN {X 0,Y 162.868,Z 308.498,A -85,B 0,C 180,E1 -23142.46,E2 -23142.46} C_VEL
LIN {X 0,Y 163.693,Z 307.279,A -85,B 0,C 180,E1 -23144.928,E2 -23144.928} C_VEL
LIN {X 0,Y 166.458,Z 303.629,A -85,B 0,C 180,E1 -23149.741,E2 -23149.741} C_VEL
LIN {X 0,Y 169.272,Z 299.728,A -85,B 0,C 180,E1 -23153.23,E2 -23153.23} C_VEL
LIN {X 0,Y 172.561,Z 294.722,A -85,B 0,C 180,E1 -23156.616,E2 -23156.616} C_VEL
LIN {X 0,Y 176.518,Z 288.471,A -85,B 0,C 180,E1 -23159.847,E2 -23159.847} C_VEL
LIN {X 0,Y 181.201,Z 280.71,A -85,B 0,C 180,E1 -23162.888,E2 -23162.888} C_VEL
LIN {X 0,Y 186.453,Z 271.023,A -85,B 0,C 180,E1 -23165.75,E2 -23165.75} C_VEL
LIN {X 0,Y 191.131,Z 261.05,A -85,B 0,C 180,E1 -23168.018,E2 -23168.018} C_VEL
LIN {X 0,Y 195.255,Z 251.208,A -85,B 0,C 180,E1 -23169.71,E2 -23169.71} C_VEL
LIN {X 0,Y 198.928,Z 240.546,A -85,B 0,C 180,E1 -23171.148,E2 -23171.148} C_VEL
LIN {X 0,Y 202.491,Z 227.731,A -85,B 0,C 180,E1 -23172.426,E2 -23172.426} C_VEL
LIN {X 0,Y 205.105,Z 215.098,A -85,B 0,C 180,E1 -23173.312,E2 -23173.312} C_VEL
LIN {X 0,Y 206.853,Z 201.747,A -85,B 0,C 180,E1 -23173.906,E2 -23173.906} C_VEL
LIN {X 0,Y 208.847,Z 171.574,A -85,B 0,C 180,E1 -23174.864,E2 -23174.864} C_VEL
LIN {X 0,Y 208.211,Z 165.369,A -85,B 0,C 180,E1 -23175.388,E2 -23175.388} C_VEL
LIN {X 0,Y 203.058,Z 152.645,A -85,B 0,C 180,E1 -23177.832,E2 -23177.832} C_VEL
LIN {X 0,Y 198.139,Z 142.284,A -85,B 0,C 180,E1 -23180.322,E2 -23180.322} C_VEL
LIN {X 0,Y 193.338,Z 133.198,A -85,B 0,C 180,E1 -23182.976,E2 -23182.976} C_VEL
LIN {X 0,Y 189.796,Z 127.132,A -85,B 0,C 180,E1 -23185.115,E2 -23185.115} C_VEL
LIN {X 0,Y 187.532,Z 123.291,A -85,B 0,C 180,E1 -23186.604,E2 -23186.604} C_VEL
LIN {X 0,Y 184.091,Z 117.83,A -85,B 0,C 180,E1 -23189.056,E2 -23189.056} C_VEL
LIN {X 0,Y 179.828,Z 111.341,A -85,B 0,C 180,E1 -23192.546,E2 -23192.546} C_VEL
LIN {X 0,Y 176.763,Z 107.144,A -85,B 0,C 180,E1 -23195.474,E2 -23195.474} C_VEL
LIN {X 0,Y 175.368,Z 105.075,A -85,B 0,C 180,E1 -23197.011,E2 -23197.011} C_VEL
LIN {X 0,Y 173.518,Z 103.132,A -85,B 0,C 180,E1 -23199.201,E2 -23199.201} C_VEL
LIN {X 0,Y 171.394,Z 100.773,A -85,B 0,C 180,E1 -23202.243,E2 -23202.243} C_VEL
LIN {X 0,Y 170.374,Z 98.365,A -85,B 0,C 180,E1 -23204.293,E2 -23204.293} C_VEL
LIN {X 0,Y 169.698,Z 97.955,A -85,B 0,C 180,E1 -23205.612,E2 -23205.612} C_VEL
LIN {X 0,Y 167.533,Z 96.687,A -85,B 0,C 180,E1 -23212.77,E2 -23212.77} C_VEL
LIN {X 0,Y 167.921,Z 96.571,A -85,B 0,C 180,E1 -23220,E2 -23220} C_VEL
LIN {X 0,Y 170.58,Z 98.229,A -85,B 0,C 180,E1 -23226.802,E2 -23226.802} C_VEL
LIN {X 0,Y 171.871,Z 101.192,A -85,B 0,C 180,E1 -23229.265,E2 -23229.265} C_VEL
LIN {X 0,Y 174.263,Z 103.474,A -85,B 0,C 180,E1 -23232.445,E2 -23232.445} C_VEL
LIN {X 0,Y 175.296,Z 104.149,A -85,B 0,C 180,E1 -23233.586,E2 -23233.586} C_VEL
LIN {X 0,Y 176.887,Z 107.062,A -85,B 0,C 180,E1 -23235.409,E2 -23235.409} C_VEL
LIN {X 0,Y 179.658,Z 109.692,A -85,B 0,C 180,E1 -23237.942,E2 -23237.942} C_VEL
LIN {X 0,Y 181.935,Z 113.072,A -85,B 0,C 180,E1 -23239.902,E2 -23239.902} C_VEL
LIN {X 0,Y 183.695,Z 114.857,A -85,B 0,C 180,E1 -23241.221,E2 -23241.221} C_VEL
LIN {X 0,Y 186.471,Z 118.651,A -85,B 0,C 180,E1 -23243.216,E2 -23243.216} C_VEL
LIN {X 0,Y 187.694,Z 120.217,A -85,B 0,C 180,E1 -23244.029,E2 -23244.029} C_VEL
LIN {X 0,Y 191.422,Z 125.425,A -85,B 0,C 180,E1 -23246.36,E2 -23246.36} C_VEL
LIN {X 0,Y 196.258,Z 132.421,A -85,B 0,C 180,E1 -23249.056,E2 -23249.056} C_VEL
LIN {X 0,Y 202.388,Z 142.225,A -85,B 0,C 180,E1 -23252.11,E2 -23252.11} C_VEL
LIN {X 0,Y 208.309,Z 152.989,A -85,B 0,C 180,E1 -23254.777,E2 -23254.777} C_VEL
LIN {X 0,Y 209.855,Z 156.007,A -85,B 0,C 180,E1 -23255.435,E2 -23255.435} C_VEL
LIN {X 0,Y 207.331,Z 190.749,A -85,B 0,C 180,E1 -23256.536,E2 -23256.536} C_VEL
LIN {X 0,Y 205.483,Z 204.239,A -85,B 0,C 180,E1 -23257.324,E2 -23257.324} C_VEL
LIN {X 0,Y 203.077,Z 216.438,A -85,B 0,C 180,E1 -23258.401,E2 -23258.401} C_VEL
LIN {X 0,Y 199.933,Z 227.9,A -85,B 0,C 180,E1 -23259.741,E2 -23259.741} C_VEL
LIN {X 0,Y 195.962,Z 239.495,A -85,B 0,C 180,E1 -23261.525,E2 -23261.525} C_VEL
LIN {X 0,Y 191.605,Z 250.069,A -85,B 0,C 180,E1 -23263.655,E2 -23263.655} C_VEL
LIN {X 0,Y 187.289,Z 259.131,A -85,B 0,C 180,E1 -23266.035,E2 -23266.035} C_VEL
LIN {X 0,Y 182.3,Z 268.097,A -85,B 0,C 180,E1 -23269.051,E2 -23269.051} C_VEL
LIN {X 0,Y 178.066,Z 275.003,A -85,B 0,C 180,E1 -23272.127,E2 -23272.127} C_VEL
LIN {X 0,Y 173.96,Z 280.863,A -85,B 0,C 180,E1 -23275.556,E2 -23275.556} C_VEL
LIN {X 0,Y 170.615,Z 285.254,A -85,B 0,C 180,E1 -23279.009,E2 -23279.009} C_VEL
LIN {X 0,Y 167.83,Z 288.532,A -85,B 0,C 180,E1 -23282.572,E2 -23282.572} C_VEL
LIN {X 0,Y 166.259,Z 290.142,A -85,B 0,C 180,E1 -23284.994,E2 -23284.994} C_VEL
LIN {X 0,Y 164.997,Z 291.337,A -85,B 0,C 180,E1 -23287.459,E2 -23287.459} C_VEL
LIN {X 0,Y 163.651,Z 292.253,A -85,B 0,C 180,E1 -23290.872,E2 -23290.872} C_VEL
LIN {X 0,Y 162.54,Z 292.373,A -85,B 0,C 180,E1 -23294.964,E2 -23294.964} C_VEL
LIN {X 0,Y 162.164,Z 291.933,A -85,B 0,C 180,E1 -23297.485,E2 -23297.485} C_VEL
LIN {X 0,Y 162.033,Z 291.053,A -85,B 0,C 180,E1 -23300.009,E2 -23300.009} C_VEL
LIN {X 0,Y 162.433,Z 288.571,A -85,B 0,C 180,E1 -23304.349,E2 -23304.349} C_VEL
LIN {X 0,Y 162.965,Z 284.728,A -85,B 0,C 180,E1 -23308.765,E2 -23308.765} C_VEL
LIN {X 0,Y 164.018,Z 280.306,A -85,B 0,C 180,E1 -23312.456,E2 -23312.456} C_VEL
LIN {X 0,Y 165.427,Z 274.711,A -85,B 0,C 180,E1 -23316.097,E2 -23316.097} C_VEL
LIN {X 0,Y 167.53,Z 267.694,A -85,B 0,C 180,E1 -23319.66,E2 -23319.66} C_VEL
LIN {X 0,Y 170.002,Z 258.944,A -85,B 0,C 180,E1 -23323.143,E2 -23323.143} C_VEL
LIN {X 0,Y 172.841,Z 248.99,A -85,B 0,C 180,E1 -23326.234,E2 -23326.234} C_VEL
LIN {X 0,Y 175.635,Z 238.782,A -85,B 0,C 180,E1 -23328.67,E2 -23328.67} C_VEL
LIN {X 0,Y 178.17,Z 227.501,A -85,B 0,C 180,E1 -23330.794,E2 -23330.794} C_VEL
LIN {X 0,Y 180.241,Z 215.842,A -85,B 0,C 180,E1 -23332.496,E2 -23332.496} C_VEL
LIN {X 0,Y 181.943,Z 203.095,A -85,B 0,C 180,E1 -23333.853,E2 -23333.853} C_VEL
LIN {X 0,Y 183.165,Z 189.525,A -85,B 0,C 180,E1 -23334.814,E2 -23334.814} C_VEL
LIN {X 0,Y 185.949,Z 132.679,A -85,B 0,C 180,E1 -23336.926,E2 -23336.926} C_VEL
LIN {X 0,Y 178.931,Z 117.621,A -85,B 0,C 180,E1 -23339.114,E2 -23339.114} C_VEL
LIN {X 0,Y 171.415,Z 104.014,A -85,B 0,C 180,E1 -23341.6,E2 -23341.6} C_VEL
LIN {X 0,Y 166.936,Z 96.811,A -85,B 0,C 180,E1 -23343.183,E2 -23343.183} C_VEL
LIN {X 0,Y 164.825,Z 93.715,A -85,B 0,C 180,E1 -23343.953,E2 -23343.953} C_VEL
LIN {X 0,Y 164.385,Z 92.005,A -85,B 0,C 180,E1 -23344.225,E2 -23344.225} C_VEL
LIN {X 0,Y 164.301,Z 92.017,A -85,B 0,C 180,E1 -23349.914,E2 -23349.914} C_VEL
LIN {X 0,Y 164.28,Z 92.021,A -85,B 0,C 180,E1 -23353.342,E2 -23353.342} C_VEL
LIN {X 0,Y 164.264,Z 92.02,A -85,B 0,C 180,E1 -23356.8,E2 -23356.8} C_VEL
LIN {X 0,Y 164.296,Z 92.012,A -85,B 0,C 180,E1 -23360.352,E2 -23360.352} C_VEL
LIN {X 0,Y 164.332,Z 92.006,A -85,B 0,C 180,E1 -23364.349,E2 -23364.349} C_VEL
LIN {X 0,Y 164.393,Z 91.999,A -85,B 0,C 180,E1 -23369.135,E2 -23369.135} C_VEL
LIN {X 0,Y 164.419,Z 91.997,A -85,B 0,C 180,E1 -23374.695,E2 -23374.695} C_VEL
LIN {X 0,Y 164.487,Z 91.987,A -85,B 0,C 180,E1 -23380.051,E2 -23380.051} C_VEL
LIN {X 0,Y 164.509,Z 91.963,A -85,B 0,C 180,E1 -23385.148,E2 -23385.148} C_VEL
LIN {X 0,Y 164.771,Z 91.96,A -85,B 0,C 180,E1 -23390.177,E2 -23390.177} C_VEL
LIN {X 0,Y 164.833,Z 91.937,A -85,B 0,C 180,E1 -23392.651,E2 -23392.651} C_VEL
LIN {X 0,Y 165.049,Z 91.901,A -85,B 0,C 180,E1 -23397.56,E2 -23397.56} C_VEL
LIN {X 0,Y 165.298,Z 91.891,A -85,B 0,C 180,E1 -23400,E2 -23400} C_VEL
LIN {X 0,Y 164.759,Z 91.954,A -85,B 0,C 180,E1 -23404.894,E2 -23404.894} C_VEL
LIN {X 0,Y 164.829,Z 91.954,A -85,B 0,C 180,E1 -23407.349,E2 -23407.349} C_VEL
LIN {X 0,Y 164.705,Z 91.962,A -85,B 0,C 180,E1 -23411.06,E2 -23411.06} C_VEL
LIN {X 0,Y 164.482,Z 91.997,A -85,B 0,C 180,E1 -23417.404,E2 -23417.404} C_VEL
LIN {X 0,Y 164.476,Z 91.992,A -85,B 0,C 180,E1 -23419.989,E2 -23419.989} C_VEL
LIN {X 0,Y 164.373,Z 92.01,A -85,B 0,C 180,E1 -23426.117,E2 -23426.117} C_VEL
LIN {X 0,Y 164.36,Z 92.015,A -85,B 0,C 180,E1 -23431.217,E2 -23431.217} C_VEL
LIN {X 0,Y 164.297,Z 92.022,A -85,B 0,C 180,E1 -23436.789,E2 -23436.789} C_VEL
LIN {X 0,Y 164.292,Z 92.018,A -85,B 0,C 180,E1 -23442.357,E2 -23442.357} C_VEL
LIN {X 0,Y 164.295,Z 92.145,A -85,B 0,C 180,E1 -23443.191,E2 -23443.191} C_VEL
LIN {X 0,Y 165.401,Z 95.978,A -85,B 0,C 180,E1 -23445.592,E2 -23445.592} C_VEL
LIN {X 0,Y 167.67,Z 100.263,A -85,B 0,C 180,E1 -23446.459,E2 -23446.459} C_VEL
LIN {X 0,Y 173.447,Z 111.77,A -85,B 0,C 180,E1 -23448.557,E2 -23448.557} C_VEL
LIN {X 0,Y 178.637,Z 123.97,A -85,B 0,C 180,E1 -23450.377,E2 -23450.377} C_VEL
LIN {X 0,Y 182.166,Z 133.691,A -85,B 0,C 180,E1 -23451.601,E2 -23451.601} C_VEL
LIN {X 0,Y 184.555,Z 161.982,A -85,B 0,C 180,E1 -23453.377,E2 -23453.377} C_VEL
LIN {X 0,Y 182.45,Z 206.13,A -85,B 0,C 180,E1 -23455.041,E2 -23455.041} C_VEL
LIN {X 0,Y 180.988,Z 220.06,A -85,B 0,C 180,E1 -23455.984,E2 -23455.984} C_VEL
LIN {X 0,Y 178.895,Z 233.002,A -85,B 0,C 180,E1 -23457.304,E2 -23457.304} C_VEL
LIN {X 0,Y 176.292,Z 245.61,A -85,B 0,C 180,E1 -23459.118,E2 -23459.118} C_VEL
LIN {X 0,Y 173.494,Z 256.84,A -85,B 0,C 180,E1 -23461.246,E2 -23461.246} C_VEL
LIN {X 0,Y 172.05,Z 262.576,A -85,B 0,C 180,E1 -23462.601,E2 -23462.601} C_VEL
LIN {X 0,Y 170.318,Z 267.123,A -85,B 0,C 180,E1 -23463.746,E2 -23463.746} C_VEL
LIN {X 0,Y 165.605,Z 274.055,A -85,B 0,C 180,E1 -23465.575,E2 -23465.575} C_VEL
LIN {X 0,Y 160.895,Z 280.387,A -85,B 0,C 180,E1 -23467.676,E2 -23467.676} C_VEL
LIN {X 0,Y 159.215,Z 284.012,A -85,B 0,C 180,E1 -23469.211,E2 -23469.211} C_VEL
LIN {X 0,Y 157.196,Z 291.472,A -85,B 0,C 180,E1 -23473.105,E2 -23473.105} C_VEL
LIN {X 0,Y 155.808,Z 297.221,A -85,B 0,C 180,E1 -23476.965,E2 -23476.965} C_VEL
LIN {X 0,Y 155.143,Z 301.748,A -85,B 0,C 180,E1 -23480.877,E2 -23480.877} C_VEL
LIN {X 0,Y 155.02,Z 305.905,A -85,B 0,C 180,E1 -23485.866,E2 -23485.866} C_VEL
LIN {X 0,Y 155.253,Z 308.116,A -85,B 0,C 180,E1 -23490,E2 -23490} C_VEL
LIN {X 0,Y 155.018,Z 309.212,A -85,B 0,C 180,E1 -23494.12,E2 -23494.12} C_VEL
LIN {X 0,Y 154.95,Z 309.326,A -85,B 0,C 180,E1 -23497.82,E2 -23497.82} C_VEL
LIN {X 0,Y 155.904,Z 308.174,A -85,B 0,C 180,E1 -23503.026,E2 -23503.026} C_VEL
LIN {X 0,Y 156.805,Z 307.003,A -85,B 0,C 180,E1 -23505.6,E2 -23505.6} C_VEL
LIN {X 0,Y 159.746,Z 303.406,A -85,B 0,C 180,E1 -23510.607,E2 -23510.607} C_VEL
LIN {X 0,Y 162.732,Z 299.562,A -85,B 0,C 180,E1 -23514.223,E2 -23514.223} C_VEL
LIN {X 0,Y 166.227,Z 294.618,A -85,B 0,C 180,E1 -23517.715,E2 -23517.715} C_VEL
LIN {X 0,Y 170.392,Z 288.434,A -85,B 0,C 180,E1 -23521.036,E2 -23521.036} C_VEL
LIN {X 0,Y 175.293,Z 280.779,A -85,B 0,C 180,E1 -23524.146,E2 -23524.146} C_VEL
LIN {X 0,Y 179.798,Z 272.974,A -85,B 0,C 180,E1 -23526.591,E2 -23526.591} C_VEL
LIN {X 0,Y 184.628,Z 263.469,A -85,B 0,C 180,E1 -23528.909,E2 -23528.909} C_VEL
LIN {X 0,Y 188.226,Z 255.529,A -85,B 0,C 180,E1 -23530.448,E2 -23530.448} C_VEL
LIN {X 0,Y 192.536,Z 244.423,A -85,B 0,C 180,E1 -23532.123,E2 -23532.123} C_VEL
LIN {X 0,Y 196.489,Z 231.988,A -85,B 0,C 180,E1 -23533.514,E2 -23533.514} C_VEL
LIN {X 0,Y 199.48,Z 219.39,A -85,B 0,C 180,E1 -23534.534,E2 -23534.534} C_VEL
LIN {X 0,Y 201.743,Z 205.617,A -85,B 0,C 180,E1 -23535.252,E2 -23535.252} C_VEL
LIN {X 0,Y 204.177,Z 173.432,A -85,B 0,C 180,E1 -23536.29,E2 -23536.29} C_VEL
LIN {X 0,Y 203.723,Z 168.4,A -85,B 0,C 180,E1 -23536.72,E2 -23536.72} C_VEL
LIN {X 0,Y 198.929,Z 156.327,A -85,B 0,C 180,E1 -23539.16,E2 -23539.16} C_VEL
LIN {X 0,Y 194.794,Z 147.371,A -85,B 0,C 180,E1 -23541.397,E2 -23541.397} C_VEL
LIN {X 0,Y 190.389,Z 138.731,A -85,B 0,C 180,E1 -23543.985,E2 -23543.985} C_VEL
LIN {X 0,Y 186.839,Z 132.363,A -85,B 0,C 180,E1 -23546.281,E2 -23546.281} C_VEL
LIN {X 0,Y 184.664,Z 128.652,A -85,B 0,C 180,E1 -23547.804,E2 -23547.804} C_VEL
LIN {X 0,Y 181.745,Z 123.806,A -85,B 0,C 180,E1 -23550.029,E2 -23550.029} C_VEL
LIN {X 0,Y 177.857,Z 117.649,A -85,B 0,C 180,E1 -23553.413,E2 -23553.413} C_VEL
LIN {X 0,Y 174.875,Z 113.276,A -85,B 0,C 180,E1 -23556.463,E2 -23556.463} C_VEL
LIN {X 0,Y 173.667,Z 111.507,A -85,B 0,C 180,E1 -23557.875,E2 -23557.875} C_VEL
LIN {X 0,Y 172.021,Z 109.827,A -85,B 0,C 180,E1 -23559.935,E2 -23559.935} C_VEL
LIN {X 0,Y 169.799,Z 106.952,A -85,B 0,C 180,E1 -23563.467,E2 -23563.467} C_VEL
LIN {X 0,Y 169.08,Z 105.078,A -85,B 0,C 180,E1 -23565.096,E2 -23565.096} C_VEL
LIN {X 0,Y 166.667,Z 103.745,A -85,B 0,C 180,E1 -23572.732,E2 -23572.732} C_VEL
LIN {X 0,Y 167.049,Z 103.617,A -85,B 0,C 180,E1 -23580,E2 -23580} C_VEL
LIN {X 0,Y 169.381,Z 105.206,A -85,B 0,C 180,E1 -23586.253,E2 -23586.253} C_VEL
LIN {X 0,Y 170.99,Z 108.516,A -85,B 0,C 180,E1 -23589.328,E2 -23589.328} C_VEL
LIN {X 0,Y 173.217,Z 110.491,A -85,B 0,C 180,E1 -23592.299,E2 -23592.299} C_VEL
LIN {X 0,Y 173.792,Z 111.077,A -85,B 0,C 180,E1 -23592.981,E2 -23592.981} C_VEL
LIN {X 0,Y 175.865,Z 114.366,A -85,B 0,C 180,E1 -23595.352,E2 -23595.352} C_VEL
LIN {X 0,Y 177.936,Z 116.421,A -85,B 0,C 180,E1 -23597.305,E2 -23597.305} C_VEL
LIN {X 0,Y 180.401,Z 119.928,A -85,B 0,C 180,E1 -23599.486,E2 -23599.486} C_VEL
LIN {X 0,Y 181.795,Z 121.533,A -85,B 0,C 180,E1 -23600.582,E2 -23600.582} C_VEL
LIN {X 0,Y 184.758,Z 125.448,A -85,B 0,C 180,E1 -23602.771,E2 -23602.771} C_VEL
LIN {X 0,Y 190.577,Z 133.811,A -85,B 0,C 180,E1 -23606.542,E2 -23606.542} C_VEL
LIN {X 0,Y 195.937,Z 142.303,A -85,B 0,C 180,E1 -23609.551,E2 -23609.551} C_VEL
LIN {X 0,Y 200.934,Z 150.861,A -85,B 0,C 180,E1 -23612.067,E2 -23612.067} C_VEL
LIN {X 0,Y 205.094,Z 158.899,A -85,B 0,C 180,E1 -23614.016,E2 -23614.016} C_VEL
LIN {X 0,Y 202.695,Z 190.84,A -85,B 0,C 180,E1 -23615.039,E2 -23615.039} C_VEL
LIN {X 0,Y 200.858,Z 204.01,A -85,B 0,C 180,E1 -23615.806,E2 -23615.806} C_VEL
LIN {X 0,Y 198.419,Z 215.989,A -85,B 0,C 180,E1 -23616.839,E2 -23616.839} C_VEL
LIN {X 0,Y 195.378,Z 227.031,A -85,B 0,C 180,E1 -23618.106,E2 -23618.106} C_VEL
LIN {X 0,Y 191.75,Z 237.546,A -85,B 0,C 180,E1 -23619.674,E2 -23619.674} C_VEL
LIN {X 0,Y 187.719,Z 247.262,A -85,B 0,C 180,E1 -23621.515,E2 -23621.515} C_VEL
LIN {X 0,Y 183.435,Z 256.399,A -85,B 0,C 180,E1 -23623.757,E2 -23623.757} C_VEL
LIN {X 0,Y 178.556,Z 265.168,A -85,B 0,C 180,E1 -23626.464,E2 -23626.464} C_VEL
LIN {X 0,Y 173.7,Z 272.959,A -85,B 0,C 180,E1 -23629.656,E2 -23629.656} C_VEL
LIN {X 0,Y 169.367,Z 279.154,A -85,B 0,C 180,E1 -23633.009,E2 -23633.009} C_VEL
LIN {X 0,Y 165.521,Z 284.029,A -85,B 0,C 180,E1 -23636.497,E2 -23636.497} C_VEL
LIN {X 0,Y 162.575,Z 287.475,A -85,B 0,C 180,E1 -23639.835,E2 -23639.835} C_VEL
LIN {X 0,Y 159.693,Z 290.39,A -85,B 0,C 180,E1 -23643.89,E2 -23643.89} C_VEL
LIN {X 0,Y 158.301,Z 291.618,A -85,B 0,C 180,E1 -23646.449,E2 -23646.449} C_VEL
LIN {X 0,Y 156.693,Z 292.659,A -85,B 0,C 180,E1 -23650.371,E2 -23650.371} C_VEL
LIN {X 0,Y 155.58,Z 292.779,A -85,B 0,C 180,E1 -23654.274,E2 -23654.274} C_VEL
LIN {X 0,Y 155.127,Z 292.373,A -85,B 0,C 180,E1 -23656.908,E2 -23656.908} C_VEL
LIN {X 0,Y 154.944,Z 291.555,A -85,B 0,C 180,E1 -23659.547,E2 -23659.547} C_VEL
LIN {X 0,Y 155.381,Z 288.636,A -85,B 0,C 180,E1 -23664.81,E2 -23664.81} C_VEL
LIN {X 0,Y 155.862,Z 285.357,A -85,B 0,C 180,E1 -23668.708,E2 -23668.708} C_VEL
LIN {X 0,Y 156.935,Z 281.008,A -85,B 0,C 180,E1 -23672.567,E2 -23672.567} C_VEL
LIN {X 0,Y 158.372,Z 275.493,A -85,B 0,C 180,E1 -23676.37,E2 -23676.37} C_VEL
LIN {X 0,Y 160.541,Z 268.594,A -85,B 0,C 180,E1 -23680.085,E2 -23680.085} C_VEL
LIN {X 0,Y 163.128,Z 259.966,A -85,B 0,C 180,E1 -23683.707,E2 -23683.707} C_VEL
LIN {X 0,Y 165.751,Z 251.12,A -85,B 0,C 180,E1 -23686.631,E2 -23686.631} C_VEL
LIN {X 0,Y 168.594,Z 241.369,A -85,B 0,C 180,E1 -23689.165,E2 -23689.165} C_VEL
LIN {X 0,Y 171.269,Z 230.684,A -85,B 0,C 180,E1 -23691.358,E2 -23691.358} C_VEL
LIN {X 0,Y 173.607,Z 218.752,A -85,B 0,C 180,E1 -23693.248,E2 -23693.248} C_VEL
LIN {X 0,Y 175.469,Z 206.354,A -85,B 0,C 180,E1 -23694.712,E2 -23694.712} C_VEL
LIN {X 0,Y 176.819,Z 193.44,A -85,B 0,C 180,E1 -23695.769,E2 -23695.769} C_VEL
LIN {X 0,Y 177.742,Z 178.575,A -85,B 0,C 180,E1 -23696.462,E2 -23696.462} C_VEL
LIN {X 0,Y 179.932,Z 134.595,A -85,B 0,C 180,E1 -23698.081,E2 -23698.081} C_VEL
LIN {X 0,Y 173.112,Z 120.087,A -85,B 0,C 180,E1 -23700.351,E2 -23700.351} C_VEL
LIN {X 0,Y 166.498,Z 108.197,A -85,B 0,C 180,E1 -23702.683,E2 -23702.683} C_VEL
LIN {X 0,Y 161.2,Z 99.881,A -85,B 0,C 180,E1 -23704.678,E2 -23704.678} C_VEL
LIN {X 0,Y 159.625,Z 97.286,A -85,B 0,C 180,E1 -23705.316,E2 -23705.316} C_VEL
LIN {X 0,Y 157.875,Z 94.924,A -85,B 0,C 180,E1 -23706.015,E2 -23706.015} C_VEL
LIN {X 0,Y 157.274,Z 92.893,A -85,B 0,C 180,E1 -23706.407,E2 -23706.407} C_VEL
LIN {X 0,Y 157.214,Z 92.897,A -85,B 0,C 180,E1 -23712.11,E2 -23712.11} C_VEL
LIN {X 0,Y 157.194,Z 92.901,A -85,B 0,C 180,E1 -23717.884,E2 -23717.884} C_VEL
LIN {X 0,Y 157.27,Z 92.887,A -85,B 0,C 180,E1 -23723.551,E2 -23723.551} C_VEL
LIN {X 0,Y 157.295,Z 92.889,A -85,B 0,C 180,E1 -23728.096,E2 -23728.096} C_VEL
LIN {X 0,Y 157.325,Z 92.885,A -85,B 0,C 180,E1 -23733.467,E2 -23733.467} C_VEL
LIN {X 0,Y 157.397,Z 92.873,A -85,B 0,C 180,E1 -23739.668,E2 -23739.668} C_VEL
LIN {X 0,Y 157.445,Z 92.836,A -85,B 0,C 180,E1 -23744.465,E2 -23744.465} C_VEL
LIN {X 0,Y 157.693,Z 92.842,A -85,B 0,C 180,E1 -23749.731,E2 -23749.731} C_VEL
LIN {X 0,Y 157.77,Z 92.82,A -85,B 0,C 180,E1 -23752.32,E2 -23752.32} C_VEL
LIN {X 0,Y 158.26,Z 92.767,A -85,B 0,C 180,E1 -23760,E2 -23760} C_VEL
LIN {X 0,Y 157.766,Z 92.833,A -85,B 0,C 180,E1 -23767.68,E2 -23767.68} C_VEL
LIN {X 0,Y 157.639,Z 92.842,A -85,B 0,C 180,E1 -23771.236,E2 -23771.236} C_VEL
LIN {X 0,Y 157.44,Z 92.867,A -85,B 0,C 180,E1 -23775.536,E2 -23775.536} C_VEL
LIN {X 0,Y 157.369,Z 92.878,A -85,B 0,C 180,E1 -23780.933,E2 -23780.933} C_VEL
LIN {X 0,Y 157.312,Z 92.892,A -85,B 0,C 180,E1 -23786.681,E2 -23786.681} C_VEL
LIN {X 0,Y 157.27,Z 92.897,A -85,B 0,C 180,E1 -23792.429,E2 -23792.429} C_VEL
LIN {X 0,Y 157.27,Z 92.897,A -85,B 0,C 180,E1 -23796.449,E2 -23796.449} C_VEL
LIN {X 0,Y 157.263,Z 92.919,A -85,B 0,C 180,E1 -23801.648,E2 -23801.648} C_VEL
LIN {X 0,Y 157.892,Z 95.341,A -85,B 0,C 180,E1 -23803.27,E2 -23803.27} C_VEL
LIN {X 0,Y 160.345,Z 99.801,A -85,B 0,C 180,E1 -23804.309,E2 -23804.309} C_VEL
LIN {X 0,Y 166.32,Z 111.257,A -85,B 0,C 180,E1 -23806.686,E2 -23806.686} C_VEL
LIN {X 0,Y 171.339,Z 122.374,A -85,B 0,C 180,E1 -23808.579,E2 -23808.579} C_VEL
LIN {X 0,Y 176.337,Z 135.629,A -85,B 0,C 180,E1 -23810.426,E2 -23810.426} C_VEL
LIN {X 0,Y 178.023,Z 156.5,A -85,B 0,C 180,E1 -23811.801,E2 -23811.801} C_VEL
LIN {X 0,Y 178.522,Z 163.796,A -85,B 0,C 180,E1 -23812.251,E2 -23812.251} C_VEL
LIN {X 0,Y 176.416,Z 205.223,A -85,B 0,C 180,E1 -23813.836,E2 -23813.836} C_VEL
LIN {X 0,Y 175.015,Z 218.568,A -85,B 0,C 180,E1 -23814.742,E2 -23814.742} C_VEL
LIN {X 0,Y 172.933,Z 231.328,A -85,B 0,C 180,E1 -23816.027,E2 -23816.027} C_VEL
LIN {X 0,Y 170.526,Z 242.643,A -85,B 0,C 180,E1 -23817.603,E2 -23817.603} C_VEL
LIN {X 0,Y 168.026,Z 253.065,A -85,B 0,C 180,E1 -23819.525,E2 -23819.525} C_VEL
LIN {X 0,Y 165.651,Z 261.657,A -85,B 0,C 180,E1 -23821.49,E2 -23821.49} C_VEL
LIN {X 0,Y 163.386,Z 269.917,A -85,B 0,C 180,E1 -23823.838,E2 -23823.838} C_VEL
LIN {X 0,Y 160.672,Z 278.444,A -85,B 0,C 180,E1 -23826.816,E2 -23826.816} C_VEL
LIN {X 0,Y 159.215,Z 284.012,A -85,B 0,C 180,E1 -23829.211,E2 -23829.211} C_VEL
LIN {X 0,Y 157.64,Z 287.475,A -85,B 0,C 180,E1 -23830.844,E2 -23830.844} C_VEL
LIN {X 0,Y 153.42,Z 292.507,A -85,B 0,C 180,E1 -23833.583,E2 -23833.583} C_VEL
LIN {X 0,Y 149.457,Z 296.901,A -85,B 0,C 180,E1 -23836.617,E2 -23836.617} C_VEL
LIN {X 0,Y 148.333,Z 299.285,A -85,B 0,C 180,E1 -23838.655,E2 -23838.655} C_VEL
LIN {X 0,Y 147.892,Z 303.578,A -85,B 0,C 180,E1 -23843.177,E2 -23843.177} C_VEL
LIN {X 0,Y 147.961,Z 306.352,A -85,B 0,C 180,E1 -23847.277,E2 -23847.277} C_VEL
LIN {X 0,Y 148.168,Z 307.646,A -85,B 0,C 180,E1 -23850,E2 -23850} C_VEL
LIN {X 0,Y 147.941,Z 308.733,A -85,B 0,C 180,E1 -23853.95,E2 -23853.95} C_VEL
LIN {X 0,Y 147.912,Z 308.953,A -85,B 0,C 180,E1 -23858.195,E2 -23858.195} C_VEL
LIN {X 0,Y 148.966,Z 307.849,A -85,B 0,C 180,E1 -23863.644,E2 -23863.644} C_VEL
LIN {X 0,Y 149.941,Z 306.722,A -85,B 0,C 180,E1 -23866.334,E2 -23866.334} C_VEL
LIN {X 0,Y 151.358,Z 305.16,A -85,B 0,C 180,E1 -23868.967,E2 -23868.967} C_VEL
LIN {X 0,Y 154.049,Z 302.053,A -85,B 0,C 180,E1 -23872.817,E2 -23872.817} C_VEL
LIN {X 0,Y 158.06,Z 296.983,A -85,B 0,C 180,E1 -23877.216,E2 -23877.216} C_VEL
LIN {X 0,Y 162.771,Z 290.606,A -85,B 0,C 180,E1 -23881.207,E2 -23881.207} C_VEL
LIN {X 0,Y 167.684,Z 283.541,A -85,B 0,C 180,E1 -23884.459,E2 -23884.459} C_VEL
LIN {X 0,Y 173.178,Z 274.745,A -85,B 0,C 180,E1 -23887.498,E2 -23887.498} C_VEL
LIN {X 0,Y 178.645,Z 264.787,A -85,B 0,C 180,E1 -23890.106,E2 -23890.106} C_VEL
LIN {X 0,Y 182.898,Z 255.906,A -85,B 0,C 180,E1 -23891.886,E2 -23891.886} C_VEL
LIN {X 0,Y 187.343,Z 245.025,A -85,B 0,C 180,E1 -23893.577,E2 -23893.577} C_VEL
LIN {X 0,Y 191.424,Z 232.843,A -85,B 0,C 180,E1 -23894.971,E2 -23894.971} C_VEL
LIN {X 0,Y 194.661,Z 220.099,A -85,B 0,C 180,E1 -23896.04,E2 -23896.04} C_VEL
LIN {X 0,Y 196.974,Z 207.254,A -85,B 0,C 180,E1 -23896.734,E2 -23896.734} C_VEL
LIN {X 0,Y 198.616,Z 188.584,A -85,B 0,C 180,E1 -23897.393,E2 -23897.393} C_VEL
LIN {X 0,Y 199.665,Z 173.839,A -85,B 0,C 180,E1 -23897.857,E2 -23897.857} C_VEL
LIN {X 0,Y 199.29,Z 171.305,A -85,B 0,C 180,E1 -23898.142,E2 -23898.142} C_VEL
LIN {X 0,Y 194.942,Z 159.976,A -85,B 0,C 180,E1 -23900.534,E2 -23900.534} C_VEL
LIN {X 0,Y 189.896,Z 148.938,A -85,B 0,C 180,E1 -23903.507,E2 -23903.507} C_VEL
LIN {X 0,Y 185.368,Z 140.081,A -85,B 0,C 180,E1 -23906.488,E2 -23906.488} C_VEL
LIN {X 0,Y 182.308,Z 134.652,A -85,B 0,C 180,E1 -23908.72,E2 -23908.72} C_VEL
LIN {X 0,Y 179.458,Z 129.801,A -85,B 0,C 180,E1 -23911.022,E2 -23911.022} C_VEL
LIN {X 0,Y 176.015,Z 124.063,A -85,B 0,C 180,E1 -23914.211,E2 -23914.211} C_VEL
LIN {X 0,Y 172.246,Z 118.242,A -85,B 0,C 180,E1 -23918.455,E2 -23918.455} C_VEL
LIN {X 0,Y 171.029,Z 116.888,A -85,B 0,C 180,E1 -23920.043,E2 -23920.043} C_VEL
LIN {X 0,Y 168.849,Z 114.214,A -85,B 0,C 180,E1 -23923.527,E2 -23923.527} C_VEL
LIN {X 0,Y 167.868,Z 112.012,A -85,B 0,C 180,E1 -23925.761,E2 -23925.761} C_VEL
LIN {X 0,Y 165.802,Z 110.801,A -85,B 0,C 180,E1 -23932.694,E2 -23932.694} C_VEL
LIN {X 0,Y 166.177,Z 110.69,A -85,B 0,C 180,E1 -23940,E2 -23940} C_VEL
LIN {X 0,Y 168.247,Z 112.239,A -85,B 0,C 180,E1 -23945.797,E2 -23945.797} C_VEL
LIN {X 0,Y 169.857,Z 115.474,A -85,B 0,C 180,E1 -23948.986,E2 -23948.986} C_VEL
LIN {X 0,Y 172.273,Z 117.769,A -85,B 0,C 180,E1 -23952.292,E2 -23952.292} C_VEL
LIN {X 0,Y 174.299,Z 121.009,A -85,B 0,C 180,E1 -23954.727,E2 -23954.727} C_VEL
LIN {X 0,Y 176.102,Z 122.909,A -85,B 0,C 180,E1 -23956.52,E2 -23956.52} C_VEL
LIN {X 0,Y 178.948,Z 126.855,A -85,B 0,C 180,E1 -23959.12,E2 -23959.12} C_VEL
LIN {X 0,Y 183.327,Z 132.961,A -85,B 0,C 180,E1 -23962.542,E2 -23962.542} C_VEL
LIN {X 0,Y 186.306,Z 137.338,A -85,B 0,C 180,E1 -23964.596,E2 -23964.596} C_VEL
LIN {X 0,Y 190.939,Z 144.534,A -85,B 0,C 180,E1 -23967.467,E2 -23967.467} C_VEL
LIN {X 0,Y 196.371,Z 153.891,A -85,B 0,C 180,E1 -23970.459,E2 -23970.459} C_VEL
LIN {X 0,Y 200.386,Z 161.609,A -85,B 0,C 180,E1 -23972.487,E2 -23972.487} C_VEL
LIN {X 0,Y 198.502,Z 187.984,A -85,B 0,C 180,E1 -23973.352,E2 -23973.352} C_VEL
LIN {X 0,Y 196.898,Z 200.69,A -85,B 0,C 180,E1 -23973.993,E2 -23973.993} C_VEL
LIN {X 0,Y 194.637,Z 212.362,A -85,B 0,C 180,E1 -23974.895,E2 -23974.895} C_VEL
LIN {X 0,Y 191.519,Z 224.252,A -85,B 0,C 180,E1 -23976.165,E2 -23976.165} C_VEL
LIN {X 0,Y 187.739,Z 235.465,A -85,B 0,C 180,E1 -23977.738,E2 -23977.738} C_VEL
LIN {X 0,Y 183.474,Z 245.682,A -85,B 0,C 180,E1 -23979.566,E2 -23979.566} C_VEL
LIN {X 0,Y 178.68,Z 255.7,A -85,B 0,C 180,E1 -23981.963,E2 -23981.963} C_VEL
LIN {X 0,Y 173.359,Z 264.969,A -85,B 0,C 180,E1 -23984.81,E2 -23984.81} C_VEL
LIN {X 0,Y 168.216,Z 272.907,A -85,B 0,C 180,E1 -23988.05,E2 -23988.05} C_VEL
LIN {X 0,Y 163.628,Z 279.187,A -85,B 0,C 180,E1 -23991.48,E2 -23991.48} C_VEL
LIN {X 0,Y 159.503,Z 284.138,A -85,B 0,C 180,E1 -23995.054,E2 -23995.054} C_VEL
LIN {X 0,Y 156.007,Z 287.965,A -85,B 0,C 180,E1 -23998.863,E2 -23998.863} C_VEL
LIN {X 0,Y 153.19,Z 290.639,A -85,B 0,C 180,E1 -24002.692,E2 -24002.692} C_VEL
LIN {X 0,Y 151.663,Z 291.899,A -85,B 0,C 180,E1 -24005.351,E2 -24005.351} C_VEL
LIN {X 0,Y 149.735,Z 293.069,A -85,B 0,C 180,E1 -24009.837,E2 -24009.837} C_VEL
LIN {X 0,Y 148.652,Z 293.185,A -85,B 0,C 180,E1 -24013.521,E2 -24013.521} C_VEL
LIN {X 0,Y 147.881,Z 292.042,A -85,B 0,C 180,E1 -24019.042,E2 -24019.042} C_VEL
LIN {X 0,Y 147.915,Z 290.829,A -85,B 0,C 180,E1 -24021.805,E2 -24021.805} C_VEL
LIN {X 0,Y 148.326,Z 288.719,A -85,B 0,C 180,E1 -24025.284,E2 -24025.284} C_VEL
LIN {X 0,Y 149.021,Z 284.702,A -85,B 0,C 180,E1 -24030,E2 -24030} C_VEL
LIN {X 0,Y 150.31,Z 280.042,A -85,B 0,C 180,E1 -24034.022,E2 -24034.022} C_VEL
LIN {X 0,Y 152.005,Z 274.162,A -85,B 0,C 180,E1 -24037.973,E2 -24037.973} C_VEL
LIN {X 0,Y 154.453,Z 266.815,A -85,B 0,C 180,E1 -24041.816,E2 -24041.816} C_VEL
LIN {X 0,Y 157.309,Z 257.718,A -85,B 0,C 180,E1 -24045.549,E2 -24045.549} C_VEL
LIN {X 0,Y 160.554,Z 247.173,A -85,B 0,C 180,E1 -24048.834,E2 -24048.834} C_VEL
LIN {X 0,Y 163.671,Z 236.409,A -85,B 0,C 180,E1 -24051.407,E2 -24051.407} C_VEL
LIN {X 0,Y 166.112,Z 225.976,A -85,B 0,C 180,E1 -24053.369,E2 -24053.369} C_VEL
LIN {X 0,Y 168.416,Z 213.466,A -85,B 0,C 180,E1 -24055.159,E2 -24055.159} C_VEL
LIN {X 0,Y 170.193,Z 200.274,A -85,B 0,C 180,E1 -24056.519,E2 -24056.519} C_VEL
LIN {X 0,Y 171.297,Z 187.154,A -85,B 0,C 180,E1 -24057.381,E2 -24057.381} C_VEL
LIN {X 0,Y 173.913,Z 136.537,A -85,B 0,C 180,E1 -24059.334,E2 -24059.334} C_VEL
LIN {X 0,Y 167.648,Z 123.179,A -85,B 0,C 180,E1 -24061.569,E2 -24061.569} C_VEL
LIN {X 0,Y 161.71,Z 112.385,A -85,B 0,C 180,E1 -24063.81,E2 -24063.81} C_VEL
LIN {X 0,Y 155.299,Z 102.208,A -85,B 0,C 180,E1 -24066.421,E2 -24066.421} C_VEL
LIN {X 0,Y 153.267,Z 98.981,A -85,B 0,C 180,E1 -24067.318,E2 -24067.318} C_VEL
LIN {X 0,Y 150.917,Z 96.094,A -85,B 0,C 180,E1 -24068.348,E2 -24068.348} C_VEL
LIN {X 0,Y 150.198,Z 93.775,A -85,B 0,C 180,E1 -24068.794,E2 -24068.794} C_VEL
LIN {X 0,Y 150.126,Z 93.778,A -85,B 0,C 180,E1 -24074.605,E2 -24074.605} C_VEL
LIN {X 0,Y 150.142,Z 93.774,A -85,B 0,C 180,E1 -24079.056,E2 -24079.056} C_VEL
LIN {X 0,Y 150.183,Z 93.775,A -85,B 0,C 180,E1 -24082.707,E2 -24082.707} C_VEL
LIN {X 0,Y 150.217,Z 93.772,A -85,B 0,C 180,E1 -24087.368,E2 -24087.368} C_VEL
LIN {X 0,Y 150.247,Z 93.77,A -85,B 0,C 180,E1 -24092.718,E2 -24092.718} C_VEL
LIN {X 0,Y 150.354,Z 93.753,A -85,B 0,C 180,E1 -24099.208,E2 -24099.208} C_VEL
LIN {X 0,Y 150.355,Z 93.716,A -85,B 0,C 180,E1 -24103.713,E2 -24103.713} C_VEL
LIN {X 0,Y 150.614,Z 93.724,A -85,B 0,C 180,E1 -24109.243,E2 -24109.243} C_VEL
LIN {X 0,Y 150.708,Z 93.701,A -85,B 0,C 180,E1 -24111.958,E2 -24111.958} C_VEL
LIN {X 0,Y 151.22,Z 93.644,A -85,B 0,C 180,E1 -24120,E2 -24120} C_VEL
LIN {X 0,Y 150.704,Z 93.711,A -85,B 0,C 180,E1 -24128.043,E2 -24128.043} C_VEL
LIN {X 0,Y 150.58,Z 93.723,A -85,B 0,C 180,E1 -24131.437,E2 -24131.437} C_VEL
LIN {X 0,Y 150.352,Z 93.752,A -85,B 0,C 180,E1 -24136.288,E2 -24136.288} C_VEL
LIN {X 0,Y 150.352,Z 93.751,A -85,B 0,C 180,E1 -24140.79,E2 -24140.79} C_VEL
LIN {X 0,Y 150.241,Z 93.774,A -85,B 0,C 180,E1 -24147.278,E2 -24147.278} C_VEL
LIN {X 0,Y 150.211,Z 93.777,A -85,B 0,C 180,E1 -24152.628,E2 -24152.628} C_VEL
LIN {X 0,Y 150.175,Z 93.78,A -85,B 0,C 180,E1 -24157.473,E2 -24157.473} C_VEL
LIN {X 0,Y 150.201,Z 93.889,A -85,B 0,C 180,E1 -24160.044,E2 -24160.044} C_VEL
LIN {X 0,Y 150.41,Z 94.87,A -85,B 0,C 180,E1 -24160.636,E2 -24160.636} C_VEL
LIN {X 0,Y 152.297,Z 98.328,A -85,B 0,C 180,E1 -24161.55,E2 -24161.55} C_VEL
LIN {X 0,Y 153.954,Z 100.997,A -85,B 0,C 180,E1 -24162.3,E2 -24162.3} C_VEL
LIN {X 0,Y 157.079,Z 106.655,A -85,B 0,C 180,E1 -24163.686,E2 -24163.686} C_VEL
LIN {X 0,Y 162.941,Z 118.332,A -85,B 0,C 180,E1 -24166.133,E2 -24166.133} C_VEL
LIN {X 0,Y 168.063,Z 130.747,A -85,B 0,C 180,E1 -24168.188,E2 -24168.188} C_VEL
LIN {X 0,Y 170.728,Z 138.61,A -85,B 0,C 180,E1 -24169.262,E2 -24169.262} C_VEL
LIN {X 0,Y 172.603,Z 164.178,A -85,B 0,C 180,E1 -24170.988,E2 -24170.988} C_VEL
LIN {X 0,Y 170.363,Z 205.401,A -85,B 0,C 180,E1 -24172.613,E2 -24172.613} C_VEL
LIN {X 0,Y 168.811,Z 219.336,A -85,B 0,C 180,E1 -24173.611,E2 -24173.611} C_VEL
LIN {X 0,Y 166.64,Z 231.758,A -85,B 0,C 180,E1 -24174.926,E2 -24174.926} C_VEL
LIN {X 0,Y 164.145,Z 242.859,A -85,B 0,C 180,E1 -24176.546,E2 -24176.546} C_VEL
LIN {X 0,Y 161.542,Z 253.173,A -85,B 0,C 180,E1 -24178.528,E2 -24178.528} C_VEL
LIN {X 0,Y 159.072,Z 261.682,A -85,B 0,C 180,E1 -24180.559,E2 -24180.559} C_VEL
LIN {X 0,Y 156.423,Z 270.787,A -85,B 0,C 180,E1 -24183.301,E2 -24183.301} C_VEL
LIN {X 0,Y 153.48,Z 279.424,A -85,B 0,C 180,E1 -24186.536,E2 -24186.536} C_VEL
LIN {X 0,Y 151.323,Z 287.288,A -85,B 0,C 180,E1 -24190.323,E2 -24190.323} C_VEL
LIN {X 0,Y 149.755,Z 292.819,A -85,B 0,C 180,E1 -24193.645,E2 -24193.645} C_VEL
LIN {X 0,Y 148.516,Z 298.226,A -85,B 0,C 180,E1 -24197.705,E2 -24197.705} C_VEL
LIN {X 0,Y 148.333,Z 299.285,A -85,B 0,C 180,E1 -24198.655,E2 -24198.655} C_VEL
LIN {X 0,Y 147.452,Z 301.47,A -85,B 0,C 180,E1 -24200.756,E2 -24200.756} C_VEL
LIN {X 0,Y 145.855,Z 303.315,A -85,B 0,C 180,E1 -24202.872,E2 -24202.872} C_VEL
LIN {X 0,Y 142.278,Z 306.084,A -85,B 0,C 180,E1 -24207.29,E2 -24207.29} C_VEL
LIN {X 0,Y 141.034,Z 307.312,A -85,B 0,C 180,E1 -24210.446,E2 -24210.446} C_VEL
LIN {X 0,Y 140.87,Z 308.258,A -85,B 0,C 180,E1 -24213.794,E2 -24213.794} C_VEL
LIN {X 0,Y 140.85,Z 308.578,A -85,B 0,C 180,E1 -24218.609,E2 -24218.609} C_VEL
LIN {X 0,Y 142.053,Z 307.525,A -85,B 0,C 180,E1 -24224.322,E2 -24224.322} C_VEL
LIN {X 0,Y 143.105,Z 306.429,A -85,B 0,C 180,E1 -24227.137,E2 -24227.137} C_VEL
LIN {X 0,Y 144.634,Z 304.913,A -85,B 0,C 180,E1 -24229.885,E2 -24229.885} C_VEL
LIN {X 0,Y 147.514,Z 301.859,A -85,B 0,C 180,E1 -24233.889,E2 -24233.889} C_VEL
LIN {X 0,Y 151.472,Z 297.212,A -85,B 0,C 180,E1 -24238.168,E2 -24238.168} C_VEL
LIN {X 0,Y 156.74,Z 290.535,A -85,B 0,C 180,E1 -24242.552,E2 -24242.552} C_VEL
LIN {X 0,Y 161.866,Z 283.566,A -85,B 0,C 180,E1 -24245.884,E2 -24245.884} C_VEL
LIN {X 0,Y 167.599,Z 274.87,A -85,B 0,C 180,E1 -24248.976,E2 -24248.976} C_VEL
LIN {X 0,Y 172.746,Z 265.992,A -85,B 0,C 180,E1 -24251.385,E2 -24251.385} C_VEL
LIN {X 0,Y 177.695,Z 256.261,A -85,B 0,C 180,E1 -24253.409,E2 -24253.409} C_VEL
LIN {X 0,Y 182.279,Z 245.622,A -85,B 0,C 180,E1 -24255.111,E2 -24255.111} C_VEL
LIN {X 0,Y 186.493,Z 233.72,A -85,B 0,C 180,E1 -24256.506,E2 -24256.506} C_VEL
LIN {X 0,Y 189.835,Z 221.373,A -85,B 0,C 180,E1 -24257.572,E2 -24257.572} C_VEL
LIN {X 0,Y 192.446,Z 208.031,A -85,B 0,C 180,E1 -24258.337,E2 -24258.337} C_VEL
LIN {X 0,Y 194.039,Z 191.946,A -85,B 0,C 180,E1 -24258.925,E2 -24258.925} C_VEL
LIN {X 0,Y 195.219,Z 174.839,A -85,B 0,C 180,E1 -24259.5,E2 -24259.5} C_VEL
LIN {X 0,Y 191.127,Z 163.87,A -85,B 0,C 180,E1 -24261.924,E2 -24261.924} C_VEL
LIN {X 0,Y 186.493,Z 153.461,A -85,B 0,C 180,E1 -24264.869,E2 -24264.869} C_VEL
LIN {X 0,Y 182.325,Z 145.086,A -85,B 0,C 180,E1 -24267.829,E2 -24267.829} C_VEL
LIN {X 0,Y 179.739,Z 140.241,A -85,B 0,C 180,E1 -24269.867,E2 -24269.867} C_VEL
LIN {X 0,Y 177.167,Z 135.655,A -85,B 0,C 180,E1 -24272.098,E2 -24272.098} C_VEL
LIN {X 0,Y 174.199,Z 130.471,A -85,B 0,C 180,E1 -24275.034,E2 -24275.034} C_VEL
LIN {X 0,Y 170.698,Z 124.775,A -85,B 0,C 180,E1 -24279.239,E2 -24279.239} C_VEL
LIN {X 0,Y 167.572,Z 120.859,A -85,B 0,C 180,E1 -24284.259,E2 -24284.259} C_VEL
LIN {X 0,Y 166.872,Z 119.099,A -85,B 0,C 180,E1 -24285.985,E2 -24285.985} C_VEL
LIN {X 0,Y 164.938,Z 117.858,A -85,B 0,C 180,E1 -24292.655,E2 -24292.655} C_VEL
LIN {X 0,Y 164.898,Z 117.566,A -85,B 0,C 180,E1 -24297.557,E2 -24297.557} C_VEL
LIN {X 0,Y 165.672,Z 118.168,A -85,B 0,C 180,E1 -24301.519,E2 -24301.519} C_VEL
LIN {X 0,Y 167.11,Z 119.213,A -85,B 0,C 180,E1 -24305.302,E2 -24305.302} C_VEL
LIN {X 0,Y 168.93,Z 122.702,A -85,B 0,C 180,E1 -24308.975,E2 -24308.975} C_VEL
LIN {X 0,Y 170.819,Z 124.546,A -85,B 0,C 180,E1 -24311.645,E2 -24311.645} C_VEL
LIN {X 0,Y 173.04,Z 127.984,A -85,B 0,C 180,E1 -24314.404,E2 -24314.404} C_VEL
LIN {X 0,Y 174.434,Z 129.592,A -85,B 0,C 180,E1 -24315.856,E2 -24315.856} C_VEL
LIN {X 0,Y 177.378,Z 133.634,A -85,B 0,C 180,E1 -24318.642,E2 -24318.642} C_VEL
LIN {X 0,Y 181.619,Z 139.944,A -85,B 0,C 180,E1 -24322.091,E2 -24322.091} C_VEL
LIN {X 0,Y 185.564,Z 146.002,A -85,B 0,C 180,E1 -24324.86,E2 -24324.86} C_VEL
LIN {X 0,Y 190.463,Z 154.302,A -85,B 0,C 180,E1 -24327.915,E2 -24327.915} C_VEL
LIN {X 0,Y 195.282,Z 163.307,A -85,B 0,C 180,E1 -24330.598,E2 -24330.598} C_VEL
LIN {X 0,Y 195.97,Z 164.727,A -85,B 0,C 180,E1 -24330.965,E2 -24330.965} C_VEL
LIN {X 0,Y 193.778,Z 191.692,A -85,B 0,C 180,E1 -24331.855,E2 -24331.855} C_VEL
LIN {X 0,Y 191.888,Z 204.441,A -85,B 0,C 180,E1 -24332.606,E2 -24332.606} C_VEL
LIN {X 0,Y 189.286,Z 216.242,A -85,B 0,C 180,E1 -24333.609,E2 -24333.609} C_VEL
LIN {X 0,Y 185.63,Z 228.548,A -85,B 0,C 180,E1 -24335.042,E2 -24335.042} C_VEL
LIN {X 0,Y 181.148,Z 240.232,A -85,B 0,C 180,E1 -24336.851,E2 -24336.851} C_VEL
LIN {X 0,Y 176.286,Z 250.694,A -85,B 0,C 180,E1 -24338.976,E2 -24338.976} C_VEL
LIN {X 0,Y 171.022,Z 260.474,A -85,B 0,C 180,E1 -24341.655,E2 -24341.655} C_VEL
LIN {X 0,Y 165.519,Z 269.03,A -85,B 0,C 180,E1 -24344.666,E2 -24344.666} C_VEL
LIN {X 0,Y 161.029,Z 275.335,A -85,B 0,C 180,E1 -24347.6,E2 -24347.6} C_VEL
LIN {X 0,Y 156.452,Z 281.04,A -85,B 0,C 180,E1 -24351.031,E2 -24351.031} C_VEL
LIN {X 0,Y 152.29,Z 285.674,A -85,B 0,C 180,E1 -24354.77,E2 -24354.77} C_VEL
LIN {X 0,Y 148.763,Z 289.16,A -85,B 0,C 180,E1 -24358.69,E2 -24358.69} C_VEL
LIN {X 0,Y 146.77,Z 290.888,A -85,B 0,C 180,E1 -24361.39,E2 -24361.39} C_VEL
LIN {X 0,Y 143.687,Z 293.071,A -85,B 0,C 180,E1 -24366.965,E2 -24366.965} C_VEL
LIN {X 0,Y 142.604,Z 293.549,A -85,B 0,C 180,E1 -24369.819,E2 -24369.819} C_VEL
LIN {X 0,Y 141.737,Z 293.592,A -85,B 0,C 180,E1 -24372.692,E2 -24372.692} C_VEL
LIN {X 0,Y 140.805,Z 292.514,A -85,B 0,C 180,E1 -24378.484,E2 -24378.484} C_VEL
LIN {X 0,Y 140.801,Z 291.36,A -85,B 0,C 180,E1 -24381.388,E2 -24381.388} C_VEL
LIN {X 0,Y 141.186,Z 289.558,A -85,B 0,C 180,E1 -24384.602,E2 -24384.602} C_VEL
LIN {X 0,Y 141.667,Z 286.607,A -85,B 0,C 180,E1 -24388.579,E2 -24388.579} C_VEL
LIN {X 0,Y 142.771,Z 282.401,A -85,B 0,C 180,E1 -24392.822,E2 -24392.822} C_VEL
LIN {X 0,Y 144.622,Z 276.035,A -85,B 0,C 180,E1 -24397.68,E2 -24397.68} C_VEL
LIN {X 0,Y 147.051,Z 269.074,A -85,B 0,C 180,E1 -24401.72,E2 -24401.72} C_VEL
LIN {X 0,Y 149.952,Z 260.37,A -85,B 0,C 180,E1 -24405.634,E2 -24405.634} C_VEL
LIN {X 0,Y 153.206,Z 250.476,A -85,B 0,C 180,E1 -24409.078,E2 -24409.078} C_VEL
LIN {X 0,Y 156.404,Z 240.367,A -85,B 0,C 180,E1 -24411.76,E2 -24411.76} C_VEL
LIN {X 0,Y 159.338,Z 229.173,A -85,B 0,C 180,E1 -24414.079,E2 -24414.079} C_VEL
LIN {X 0,Y 161.905,Z 216.66,A -85,B 0,C 180,E1 -24416.073,E2 -24416.073} C_VEL
LIN {X 0,Y 163.859,Z 203.751,A -85,B 0,C 180,E1 -24417.543,E2 -24417.543} C_VEL
LIN {X 0,Y 165.243,Z 190.139,A -85,B 0,C 180,E1 -24418.572,E2 -24418.572} C_VEL
LIN {X 0,Y 168.048,Z 138.646,A -85,B 0,C 180,E1 -24420.649,E2 -24420.649} C_VEL
LIN {X 0,Y 161.866,Z 125.408,A -85,B 0,C 180,E1 -24423.029,E2 -24423.029} C_VEL
LIN {X 0,Y 155.926,Z 114.756,A -85,B 0,C 180,E1 -24425.45,E2 -24425.45} C_VEL
LIN {X 0,Y 150.986,Z 106.983,A -85,B 0,C 180,E1 -24427.616,E2 -24427.616} C_VEL
LIN {X 0,Y 148.572,Z 103.444,A -85,B 0,C 180,E1 -24428.74,E2 -24428.74} C_VEL
LIN {X 0,Y 146.543,Z 100.397,A -85,B 0,C 180,E1 -24429.735,E2 -24429.735} C_VEL
LIN {X 0,Y 145.758,Z 99.346,A -85,B 0,C 180,E1 -24430.123,E2 -24430.123} C_VEL
LIN {X 0,Y 143.848,Z 97.027,A -85,B 0,C 180,E1 -24431.08,E2 -24431.08} C_VEL
LIN {X 0,Y 143.114,Z 94.651,A -85,B 0,C 180,E1 -24431.657,E2 -24431.657} C_VEL
LIN {X 0,Y 143.058,Z 94.663,A -85,B 0,C 180,E1 -24437.469,E2 -24437.469} C_VEL
LIN {X 0,Y 143.08,Z 94.66,A -85,B 0,C 180,E1 -24441.806,E2 -24441.806} C_VEL
LIN {X 0,Y 143.184,Z 94.648,A -85,B 0,C 180,E1 -24447.322,E2 -24447.322} C_VEL
LIN {X 0,Y 143.193,Z 94.648,A -85,B 0,C 180,E1 -24452.063,E2 -24452.063} C_VEL
LIN {X 0,Y 143.279,Z 94.636,A -85,B 0,C 180,E1 -24458.746,E2 -24458.746} C_VEL
LIN {X 0,Y 143.298,Z 94.595,A -85,B 0,C 180,E1 -24462.887,E2 -24462.887} C_VEL
LIN {X 0,Y 143.54,Z 94.604,A -85,B 0,C 180,E1 -24468.706,E2 -24468.706} C_VEL
LIN {X 0,Y 143.629,Z 94.585,A -85,B 0,C 180,E1 -24471.559,E2 -24471.559} C_VEL
LIN {X 0,Y 144.179,Z 94.521,A -85,B 0,C 180,E1 -24480,E2 -24480} C_VEL
LIN {X 0,Y 143.626,Z 94.592,A -85,B 0,C 180,E1 -24488.442,E2 -24488.442} C_VEL
LIN {X 0,Y 143.507,Z 94.604,A -85,B 0,C 180,E1 -24491.628,E2 -24491.628} C_VEL
LIN {X 0,Y 143.296,Z 94.634,A -85,B 0,C 180,E1 -24497.114,E2 -24497.114} C_VEL
LIN {X 0,Y 143.277,Z 94.634,A -85,B 0,C 180,E1 -24501.252,E2 -24501.252} C_VEL
LIN {X 0,Y 143.185,Z 94.652,A -85,B 0,C 180,E1 -24507.931,E2 -24507.931} C_VEL
LIN {X 0,Y 143.162,Z 94.655,A -85,B 0,C 180,E1 -24513.43,E2 -24513.43} C_VEL
LIN {X 0,Y 143.133,Z 94.657,A -85,B 0,C 180,E1 -24517.678,E2 -24517.678} C_VEL
LIN {X 0,Y 143.965,Z 97.231,A -85,B 0,C 180,E1 -24518.236,E2 -24518.236} C_VEL
LIN {X 0,Y 145.93,Z 99.474,A -85,B 0,C 180,E1 -24519.206,E2 -24519.206} C_VEL
LIN {X 0,Y 149.835,Z 105.958,A -85,B 0,C 180,E1 -24521.151,E2 -24521.151} C_VEL
LIN {X 0,Y 154.255,Z 114.234,A -85,B 0,C 180,E1 -24523.223,E2 -24523.223} C_VEL
LIN {X 0,Y 159.311,Z 125.052,A -85,B 0,C 180,E1 -24525.458,E2 -24525.458} C_VEL
LIN {X 0,Y 164.127,Z 137.612,A -85,B 0,C 180,E1 -24527.522,E2 -24527.522} C_VEL
LIN {X 0,Y 165.106,Z 140.875,A -85,B 0,C 180,E1 -24527.958,E2 -24527.958} C_VEL
LIN {X 0,Y 166.748,Z 164.01,A -85,B 0,C 180,E1 -24529.601,E2 -24529.601} C_VEL
LIN {X 0,Y 164.468,Z 204.889,A -85,B 0,C 180,E1 -24531.261,E2 -24531.261} C_VEL
LIN {X 0,Y 162.865,Z 218.645,A -85,B 0,C 180,E1 -24532.26,E2 -24532.26} C_VEL
LIN {X 0,Y 160.642,Z 231.112,A -85,B 0,C 180,E1 -24533.604,E2 -24533.604} C_VEL
LIN {X 0,Y 157.825,Z 243.073,A -85,B 0,C 180,E1 -24535.405,E2 -24535.405} C_VEL
LIN {X 0,Y 155.116,Z 253.278,A -85,B 0,C 180,E1 -24537.45,E2 -24537.45} C_VEL
LIN {X 0,Y 152.536,Z 261.703,A -85,B 0,C 180,E1 -24539.547,E2 -24539.547} C_VEL
LIN {X 0,Y 149.47,Z 271.644,A -85,B 0,C 180,E1 -24542.713,E2 -24542.713} C_VEL
LIN {X 0,Y 146.646,Z 279.426,A -85,B 0,C 180,E1 -24545.802,E2 -24545.802} C_VEL
LIN {X 0,Y 144.563,Z 286.508,A -85,B 0,C 180,E1 -24549.362,E2 -24549.362} C_VEL
LIN {X 0,Y 142.918,Z 292.115,A -85,B 0,C 180,E1 -24552.839,E2 -24552.839} C_VEL
LIN {X 0,Y 141.554,Z 297.586,A -85,B 0,C 180,E1 -24557.09,E2 -24557.09} C_VEL
LIN {X 0,Y 140.907,Z 301.849,A -85,B 0,C 180,E1 -24561.394,E2 -24561.394} C_VEL
LIN {X 0,Y 140.869,Z 305.336,A -85,B 0,C 180,E1 -24566.209,E2 -24566.209} C_VEL
LIN {X 0,Y 141.034,Z 307.312,A -85,B 0,C 180,E1 -24570.446,E2 -24570.446} C_VEL
LIN {X 0,Y 140.578,Z 307.813,A -85,B 0,C 180,E1 -24572.027,E2 -24572.027} C_VEL
LIN {X 0,Y 139.103,Z 308.256,A -85,B 0,C 180,E1 -24574.374,E2 -24574.374} C_VEL
LIN {X 0,Y 135.061,Z 308.193,A -85,B 0,C 180,E1 -24579.965,E2 -24579.965} C_VEL
LIN {X 0,Y 134.482,Z 307.821,A -85,B 0,C 180,E1 -24582.479,E2 -24582.479} C_VEL
LIN {X 0,Y 134.611,Z 307.606,A -85,B 0,C 180,E1 -24583.319,E2 -24583.319} C_VEL
LIN {X 0,Y 136.305,Z 306.13,A -85,B 0,C 180,E1 -24588.021,E2 -24588.021} C_VEL
LIN {X 0,Y 137.955,Z 304.664,A -85,B 0,C 180,E1 -24590.892,E2 -24590.892} C_VEL
LIN {X 0,Y 141.039,Z 301.654,A -85,B 0,C 180,E1 -24595.059,E2 -24595.059} C_VEL
LIN {X 0,Y 144.889,Z 297.474,A -85,B 0,C 180,E1 -24599.177,E2 -24599.177} C_VEL
LIN {X 0,Y 149.946,Z 291.483,A -85,B 0,C 180,E1 -24603.417,E2 -24603.417} C_VEL
LIN {X 0,Y 155.237,Z 284.815,A -85,B 0,C 180,E1 -24606.86,E2 -24606.86} C_VEL
LIN {X 0,Y 161.122,Z 276.569,A -85,B 0,C 180,E1 -24610.045,E2 -24610.045} C_VEL
LIN {X 0,Y 166.35,Z 268.158,A -85,B 0,C 180,E1 -24612.53,E2 -24612.53} C_VEL
LIN {X 0,Y 172.024,Z 257.798,A -85,B 0,C 180,E1 -24614.809,E2 -24614.809} C_VEL
LIN {X 0,Y 177.354,Z 246.153,A -85,B 0,C 180,E1 -24616.731,E2 -24616.731} C_VEL
LIN {X 0,Y 181.701,Z 234.602,A -85,B 0,C 180,E1 -24618.122,E2 -24618.122} C_VEL
LIN {X 0,Y 185.151,Z 222.643,A -85,B 0,C 180,E1 -24619.182,E2 -24619.182} C_VEL
LIN {X 0,Y 187.951,Z 209.402,A -85,B 0,C 180,E1 -24619.977,E2 -24619.977} C_VEL
LIN {X 0,Y 189.494,Z 196.558,A -85,B 0,C 180,E1 -24620.497,E2 -24620.497} C_VEL
LIN {X 0,Y 190.965,Z 177.478,A -85,B 0,C 180,E1 -24621.101,E2 -24621.101} C_VEL
LIN {X 0,Y 187.268,Z 167.396,A -85,B 0,C 180,E1 -24623.473,E2 -24623.473} C_VEL
LIN {X 0,Y 182.422,Z 156.178,A -85,B 0,C 180,E1 -24626.866,E2 -24626.866} C_VEL
LIN {X 0,Y 178.052,Z 147.248,A -85,B 0,C 180,E1 -24630.354,E2 -24630.354} C_VEL
LIN {X 0,Y 175.067,Z 141.748,A -85,B 0,C 180,E1 -24633.075,E2 -24633.075} C_VEL
LIN {X 0,Y 172.364,Z 136.784,A -85,B 0,C 180,E1 -24635.937,E2 -24635.937} C_VEL
LIN {X 0,Y 169.207,Z 131.388,A -85,B 0,C 180,E1 -24640,E2 -24640} C_VEL
LIN {X 0,Y 166.386,Z 127.648,A -85,B 0,C 180,E1 -24644.849,E2 -24644.849} C_VEL
LIN {X 0,Y 165.739,Z 125.993,A -85,B 0,C 180,E1 -24646.56,E2 -24646.56} C_VEL
LIN {X 0,Y 164.074,Z 124.893,A -85,B 0,C 180,E1 -24652.617,E2 -24652.617} C_VEL
LIN {X 0,Y 164.191,Z 124.703,A -85,B 0,C 180,E1 -24658.773,E2 -24658.773} C_VEL
LIN {X 0,Y 166.011,Z 126.201,A -85,B 0,C 180,E1 -24664.857,E2 -24664.857} C_VEL
LIN {X 0,Y 167.865,Z 129.714,A -85,B 0,C 180,E1 -24668.729,E2 -24668.729} C_VEL
LIN {X 0,Y 169.438,Z 131.398,A -85,B 0,C 180,E1 -24671.06,E2 -24671.06} C_VEL
LIN {X 0,Y 171.898,Z 135.075,A -85,B 0,C 180,E1 -24674.2,E2 -24674.2} C_VEL
LIN {X 0,Y 172.758,Z 136.215,A -85,B 0,C 180,E1 -24675.144,E2 -24675.144} C_VEL
LIN {X 0,Y 176.275,Z 141.4,A -85,B 0,C 180,E1 -24678.6,E2 -24678.6} C_VEL
LIN {X 0,Y 179.26,Z 145.902,A -85,B 0,C 180,E1 -24681.112,E2 -24681.112} C_VEL
LIN {X 0,Y 183.126,Z 152.093,A -85,B 0,C 180,E1 -24683.989,E2 -24683.989} C_VEL
LIN {X 0,Y 187.991,Z 160.615,A -85,B 0,C 180,E1 -24687.18,E2 -24687.18} C_VEL
LIN {X 0,Y 191.698,Z 167.888,A -85,B 0,C 180,E1 -24689.377,E2 -24689.377} C_VEL
LIN {X 0,Y 189.505,Z 192.586,A -85,B 0,C 180,E1 -24690.175,E2 -24690.175} C_VEL
LIN {X 0,Y 187.456,Z 205.562,A -85,B 0,C 180,E1 -24690.95,E2 -24690.95} C_VEL
LIN {X 0,Y 184.792,Z 217.059,A -85,B 0,C 180,E1 -24691.944,E2 -24691.944} C_VEL
LIN {X 0,Y 180.93,Z 229.427,A -85,B 0,C 180,E1 -24693.404,E2 -24693.404} C_VEL
LIN {X 0,Y 176.316,Z 240.928,A -85,B 0,C 180,E1 -24695.2,E2 -24695.2} C_VEL
LIN {X 0,Y 171.258,Z 251.324,A -85,B 0,C 180,E1 -24697.335,E2 -24697.335} C_VEL
LIN {X 0,Y 166.555,Z 259.815,A -85,B 0,C 180,E1 -24699.659,E2 -24699.659} C_VEL
LIN {X 0,Y 161.473,Z 267.524,A -85,B 0,C 180,E1 -24702.276,E2 -24702.276} C_VEL
LIN {X 0,Y 155.713,Z 275.292,A -85,B 0,C 180,E1 -24705.787,E2 -24705.787} C_VEL
LIN {X 0,Y 150.879,Z 281.079,A -85,B 0,C 180,E1 -24709.298,E2 -24709.298} C_VEL
LIN {X 0,Y 146.404,Z 285.788,A -85,B 0,C 180,E1 -24713.126,E2 -24713.126} C_VEL
LIN {X 0,Y 142.608,Z 289.344,A -85,B 0,C 180,E1 -24717.173,E2 -24717.173} C_VEL
LIN {X 0,Y 140.442,Z 291.137,A -85,B 0,C 180,E1 -24719.972,E2 -24719.972} C_VEL
LIN {X 0,Y 137.042,Z 293.384,A -85,B 0,C 180,E1 -24725.778,E2 -24725.778} C_VEL
LIN {X 0,Y 135.815,Z 293.909,A -85,B 0,C 180,E1 -24728.763,E2 -24728.763} C_VEL
LIN {X 0,Y 134.842,Z 293.999,A -85,B 0,C 180,E1 -24731.777,E2 -24731.777} C_VEL
LIN {X 0,Y 133.752,Z 292.982,A -85,B 0,C 180,E1 -24737.867,E2 -24737.867} C_VEL
LIN {X 0,Y 133.689,Z 291.884,A -85,B 0,C 180,E1 -24740.926,E2 -24740.926} C_VEL
LIN {X 0,Y 134.094,Z 289.858,A -85,B 0,C 180,E1 -24744.752,E2 -24744.752} C_VEL
LIN {X 0,Y 134.805,Z 285.99,A -85,B 0,C 180,E1 -24750,E2 -24750} C_VEL
LIN {X 0,Y 136.148,Z 281.486,A -85,B 0,C 180,E1 -24754.441,E2 -24754.441} C_VEL
LIN {X 0,Y 138.373,Z 274.679,A -85,B 0,C 180,E1 -24759.502,E2 -24759.502} C_VEL
LIN {X 0,Y 141.119,Z 267.278,A -85,B 0,C 180,E1 -24763.684,E2 -24763.684} C_VEL
LIN {X 0,Y 143.737,Z 259.758,A -85,B 0,C 180,E1 -24767.06,E2 -24767.06} C_VEL
LIN {X 0,Y 146.885,Z 250.638,A -85,B 0,C 180,E1 -24770.298,E2 -24770.298} C_VEL
LIN {X 0,Y 150.225,Z 240.463,A -85,B 0,C 180,E1 -24773.068,E2 -24773.068} C_VEL
LIN {X 0,Y 153.318,Z 229.202,A -85,B 0,C 180,E1 -24775.452,E2 -24775.452} C_VEL
LIN {X 0,Y 155.629,Z 218.572,A -85,B 0,C 180,E1 -24777.209,E2 -24777.209} C_VEL
LIN {X 0,Y 157.776,Z 205.718,A -85,B 0,C 180,E1 -24778.793,E2 -24778.793} C_VEL
LIN {X 0,Y 159.225,Z 192.784,A -85,B 0,C 180,E1 -24779.858,E2 -24779.858} C_VEL
LIN {X 0,Y 160.475,Z 173.229,A -85,B 0,C 180,E1 -24780.757,E2 -24780.757} C_VEL
LIN {X 0,Y 162.345,Z 140.86,A -85,B 0,C 180,E1 -24782.035,E2 -24782.035} C_VEL
LIN {X 0,Y 156.219,Z 127.8,A -85,B 0,C 180,E1 -24784.575,E2 -24784.575} C_VEL
LIN {X 0,Y 150.982,Z 118.476,A -85,B 0,C 180,E1 -24786.88,E2 -24786.88} C_VEL
LIN {X 0,Y 146.695,Z 111.65,A -85,B 0,C 180,E1 -24788.906,E2 -24788.906} C_VEL
LIN {X 0,Y 141.91,Z 104.645,A -85,B 0,C 180,E1 -24791.359,E2 -24791.359} C_VEL
LIN {X 0,Y 139.775,Z 101.583,A -85,B 0,C 180,E1 -24792.541,E2 -24792.541} C_VEL
LIN {X 0,Y 139.278,Z 100.667,A -85,B 0,C 180,E1 -24792.841,E2 -24792.841} C_VEL
LIN {X 0,Y 137.016,Z 98.44,A -85,B 0,C 180,E1 -24794.102,E2 -24794.102} C_VEL
LIN {X 0,Y 136.032,Z 96.039,A -85,B 0,C 180,E1 -24794.791,E2 -24794.791} C_VEL
LIN {X 0,Y 135.969,Z 95.539,A -85,B 0,C 180,E1 -24794.949,E2 -24794.949} C_VEL
LIN {X 0,Y 136.031,Z 95.533,A -85,B 0,C 180,E1 -24800.803,E2 -24800.803} C_VEL
LIN {X 0,Y 136.087,Z 95.526,A -85,B 0,C 180,E1 -24805.721,E2 -24805.721} C_VEL
LIN {X 0,Y 136.149,Z 95.526,A -85,B 0,C 180,E1 -24812.317,E2 -24812.317} C_VEL
LIN {X 0,Y 136.246,Z 95.511,A -85,B 0,C 180,E1 -24818.834,E2 -24818.834} C_VEL
LIN {X 0,Y 136.266,Z 95.473,A -85,B 0,C 180,E1 -24825.056,E2 -24825.056} C_VEL
LIN {X 0,Y 136.434,Z 95.486,A -85,B 0,C 180,E1 -24828.165,E2 -24828.165} C_VEL
LIN {X 0,Y 136.554,Z 95.469,A -85,B 0,C 180,E1 -24831.118,E2 -24831.118} C_VEL
LIN {X 0,Y 137.136,Z 95.398,A -85,B 0,C 180,E1 -24840,E2 -24840} C_VEL
LIN {X 0,Y 136.552,Z 95.47,A -85,B 0,C 180,E1 -24848.883,E2 -24848.883} C_VEL
LIN {X 0,Y 136.443,Z 95.486,A -85,B 0,C 180,E1 -24851.89,E2 -24851.89} C_VEL
LIN {X 0,Y 136.239,Z 95.516,A -85,B 0,C 180,E1 -24858.03,E2 -24858.03} C_VEL
LIN {X 0,Y 136.198,Z 95.518,A -85,B 0,C 180,E1 -24861.746,E2 -24861.746} C_VEL
LIN {X 0,Y 136.095,Z 95.535,A -85,B 0,C 180,E1 -24868.61,E2 -24868.61} C_VEL
LIN {X 0,Y 136.063,Z 95.626,A -85,B 0,C 180,E1 -24874.447,E2 -24874.447} C_VEL
LIN {X 0,Y 137,Z 98.322,A -85,B 0,C 180,E1 -24875.136,E2 -24875.136} C_VEL
LIN {X 0,Y 139.22,Z 100.612,A -85,B 0,C 180,E1 -24876.382,E2 -24876.382} C_VEL
LIN {X 0,Y 141.792,Z 104.542,A -85,B 0,C 180,E1 -24877.834,E2 -24877.834} C_VEL
LIN {X 0,Y 143.192,Z 106.444,A -85,B 0,C 180,E1 -24878.57,E2 -24878.57} C_VEL
LIN {X 0,Y 146.159,Z 111.681,A -85,B 0,C 180,E1 -24880.139,E2 -24880.139} C_VEL
LIN {X 0,Y 150.091,Z 119.32,A -85,B 0,C 180,E1 -24882.111,E2 -24882.111} C_VEL
LIN {X 0,Y 154.707,Z 129.553,A -85,B 0,C 180,E1 -24884.304,E2 -24884.304} C_VEL
LIN {X 0,Y 158.944,Z 140.969,A -85,B 0,C 180,E1 -24886.263,E2 -24886.263} C_VEL
LIN {X 0,Y 159.623,Z 143.645,A -85,B 0,C 180,E1 -24886.61,E2 -24886.61} C_VEL
LIN {X 0,Y 160.982,Z 164.819,A -85,B 0,C 180,E1 -24888.165,E2 -24888.165} C_VEL
LIN {X 0,Y 158.666,Z 204.424,A -85,B 0,C 180,E1 -24889.813,E2 -24889.813} C_VEL
LIN {X 0,Y 156.982,Z 218.195,A -85,B 0,C 180,E1 -24890.83,E2 -24890.83} C_VEL
LIN {X 0,Y 154.739,Z 230.459,A -85,B 0,C 180,E1 -24892.182,E2 -24892.182} C_VEL
LIN {X 0,Y 152.022,Z 241.695,A -85,B 0,C 180,E1 -24893.882,E2 -24893.882} C_VEL
LIN {X 0,Y 148.749,Z 253.383,A -85,B 0,C 180,E1 -24896.278,E2 -24896.278} C_VEL
LIN {X 0,Y 146.056,Z 261.724,A -85,B 0,C 180,E1 -24898.446,E2 -24898.446} C_VEL
LIN {X 0,Y 143.119,Z 270.691,A -85,B 0,C 180,E1 -24901.394,E2 -24901.394} C_VEL
LIN {X 0,Y 140.188,Z 278.576,A -85,B 0,C 180,E1 -24904.61,E2 -24904.61} C_VEL
LIN {X 0,Y 137.878,Z 285.731,A -85,B 0,C 180,E1 -24908.312,E2 -24908.312} C_VEL
LIN {X 0,Y 135.804,Z 292.435,A -85,B 0,C 180,E1 -24912.688,E2 -24912.688} C_VEL
LIN {X 0,Y 134.261,Z 298.524,A -85,B 0,C 180,E1 -24917.913,E2 -24917.913} C_VEL
LIN {X 0,Y 133.754,Z 302.472,A -85,B 0,C 180,E1 -24922.451,E2 -24922.451} C_VEL
LIN {X 0,Y 133.787,Z 305.356,A -85,B 0,C 180,E1 -24926.989,E2 -24926.989} C_VEL
LIN {X 0,Y 133.964,Z 306.809,A -85,B 0,C 180,E1 -24930.351,E2 -24930.351} C_VEL
LIN {X 0,Y 133.81,Z 307.775,A -85,B 0,C 180,E1 -24933.688,E2 -24933.688} C_VEL
LIN {X 0,Y 133.814,Z 308.204,A -85,B 0,C 180,E1 -24939.065,E2 -24939.065} C_VEL
LIN {X 0,Y 134.611,Z 307.606,A -85,B 0,C 180,E1 -24943.319,E2 -24943.319} C_VEL
LIN {X 0,Y 134.756,Z 306.975,A -85,B 0,C 180,E1 -24945.819,E2 -24945.819} C_VEL
LIN {X 0,Y 133.797,Z 305.374,A -85,B 0,C 180,E1 -24949.983,E2 -24949.983} C_VEL
LIN {X 0,Y 133.535,Z 303.106,A -85,B 0,C 180,E1 -24954.118,E2 -24954.118} C_VEL
LIN {X 0,Y 134.735,Z 301.332,A -85,B 0,C 180,E1 -24956.468,E2 -24956.468} C_VEL
LIN {X 0,Y 138.564,Z 297.466,A -85,B 0,C 180,E1 -24960.478,E2 -24960.478} C_VEL
LIN {X 0,Y 143.208,Z 292.387,A -85,B 0,C 180,E1 -24964.359,E2 -24964.359} C_VEL
LIN {X 0,Y 148.662,Z 286.049,A -85,B 0,C 180,E1 -24967.921,E2 -24967.921} C_VEL
LIN {X 0,Y 154.693,Z 278.147,A -85,B 0,C 180,E1 -24971.206,E2 -24971.206} C_VEL
LIN {X 0,Y 160.122,Z 270.124,A -85,B 0,C 180,E1 -24973.732,E2 -24973.732} C_VEL
LIN {X 0,Y 165.848,Z 260.363,A -85,B 0,C 180,E1 -24976.087,E2 -24976.087} C_VEL
LIN {X 0,Y 171.34,Z 249.513,A -85,B 0,C 180,E1 -24978.026,E2 -24978.026} C_VEL
LIN {X 0,Y 176.413,Z 237.153,A -85,B 0,C 180,E1 -24979.633,E2 -24979.633} C_VEL
LIN {X 0,Y 180.303,Z 225.061,A -85,B 0,C 180,E1 -24980.779,E2 -24980.779} C_VEL
LIN {X 0,Y 183.35,Z 212.108,A -85,B 0,C 180,E1 -24981.629,E2 -24981.629} C_VEL
LIN {X 0,Y 185.232,Z 199.025,A -85,B 0,C 180,E1 -24982.201,E2 -24982.201} C_VEL
LIN {X 0,Y 186.784,Z 180.072,A -85,B 0,C 180,E1 -24982.816,E2 -24982.816} C_VEL
LIN {X 0,Y 183.616,Z 171.152,A -85,B 0,C 180,E1 -24985.044,E2 -24985.044} C_VEL
LIN {X 0,Y 179.422,Z 161.037,A -85,B 0,C 180,E1 -24988.24,E2 -24988.24} C_VEL
LIN {X 0,Y 175.702,Z 153.042,A -85,B 0,C 180,E1 -24991.449,E2 -24991.449} C_VEL
LIN {X 0,Y 172.879,Z 147.624,A -85,B 0,C 180,E1 -24994.218,E2 -24994.218} C_VEL
LIN {X 0,Y 170.611,Z 143.175,A -85,B 0,C 180,E1 -24996.811,E2 -24996.811} C_VEL
LIN {X 0,Y 167.871,Z 138.141,A -85,B 0,C 180,E1 -25000.591,E2 -25000.591} C_VEL
LIN {X 0,Y 165.187,Z 134.366,A -85,B 0,C 180,E1 -25005.525,E2 -25005.525} C_VEL
LIN {X 0,Y 164.592,Z 132.931,A -85,B 0,C 180,E1 -25007.202,E2 -25007.202} C_VEL
LIN {X 0,Y 163.207,Z 131.95,A -85,B 0,C 180,E1 -25012.577,E2 -25012.577} C_VEL
LIN {X 0,Y 163.318,Z 131.75,A -85,B 0,C 180,E1 -25018.767,E2 -25018.767} C_VEL
LIN {X 0,Y 164.934,Z 133.177,A -85,B 0,C 180,E1 -25024.429,E2 -25024.429} C_VEL
LIN {X 0,Y 166.692,Z 136.608,A -85,B 0,C 180,E1 -25028.295,E2 -25028.295} C_VEL
LIN {X 0,Y 168.097,Z 138.248,A -85,B 0,C 180,E1 -25030.492,E2 -25030.492} C_VEL
LIN {X 0,Y 170.512,Z 141.859,A -85,B 0,C 180,E1 -25033.709,E2 -25033.709} C_VEL
LIN {X 0,Y 174.178,Z 147.497,A -85,B 0,C 180,E1 -25037.615,E2 -25037.615} C_VEL
LIN {X 0,Y 177.834,Z 153.23,A -85,B 0,C 180,E1 -25040.835,E2 -25040.835} C_VEL
LIN {X 0,Y 182.159,Z 160.637,A -85,B 0,C 180,E1 -25044.125,E2 -25044.125} C_VEL
LIN {X 0,Y 187.157,Z 170.264,A -85,B 0,C 180,E1 -25047.459,E2 -25047.459} C_VEL
LIN {X 0,Y 187.502,Z 170.984,A -85,B 0,C 180,E1 -25047.675,E2 -25047.675} C_VEL
LIN {X 0,Y 185.389,Z 193.641,A -85,B 0,C 180,E1 -25048.431,E2 -25048.431} C_VEL
LIN {X 0,Y 183.211,Z 206.562,A -85,B 0,C 180,E1 -25049.206,E2 -25049.206} C_VEL
LIN {X 0,Y 180.63,Z 217.287,A -85,B 0,C 180,E1 -25050.146,E2 -25050.146} C_VEL
LIN {X 0,Y 176.768,Z 229.296,A -85,B 0,C 180,E1 -25051.541,E2 -25051.541} C_VEL
LIN {X 0,Y 172.251,Z 240.314,A -85,B 0,C 180,E1 -25053.236,E2 -25053.236} C_VEL
LIN {X 0,Y 167.525,Z 249.814,A -85,B 0,C 180,E1 -25055.109,E2 -25055.109} C_VEL
LIN {X 0,Y 162.508,Z 258.711,A -85,B 0,C 180,E1 -25057.432,E2 -25057.432} C_VEL
LIN {X 0,Y 156.667,Z 267.386,A -85,B 0,C 180,E1 -25060.305,E2 -25060.305} C_VEL
LIN {X 0,Y 150.78,Z 275.024,A -85,B 0,C 180,E1 -25063.741,E2 -25063.741} C_VEL
LIN {X 0,Y 145.452,Z 281.118,A -85,B 0,C 180,E1 -25067.432,E2 -25067.432} C_VEL
LIN {X 0,Y 140.635,Z 285.903,A -85,B 0,C 180,E1 -25071.342,E2 -25071.342} C_VEL
LIN {X 0,Y 136.548,Z 289.529,A -85,B 0,C 180,E1 -25075.517,E2 -25075.517} C_VEL
LIN {X 0,Y 134.189,Z 291.379,A -85,B 0,C 180,E1 -25078.417,E2 -25078.417} C_VEL
LIN {X 0,Y 132.163,Z 292.745,A -85,B 0,C 180,E1 -25081.407,E2 -25081.407} C_VEL
LIN {X 0,Y 129.067,Z 294.256,A -85,B 0,C 180,E1 -25087.594,E2 -25087.594} C_VEL
LIN {X 0,Y 127.982,Z 294.406,A -85,B 0,C 180,E1 -25090.763,E2 -25090.763} C_VEL
LIN {X 0,Y 126.728,Z 293.449,A -85,B 0,C 180,E1 -25097.184,E2 -25097.184} C_VEL
LIN {X 0,Y 126.584,Z 292.387,A -85,B 0,C 180,E1 -25100.412,E2 -25100.412} C_VEL
LIN {X 0,Y 127.012,Z 290.182,A -85,B 0,C 180,E1 -25104.871,E2 -25104.871} C_VEL
LIN {X 0,Y 127.703,Z 286.613,A -85,B 0,C 180,E1 -25110,E2 -25110} C_VEL
LIN {X 0,Y 129.077,Z 282.18,A -85,B 0,C 180,E1 -25114.685,E2 -25114.685} C_VEL
LIN {X 0,Y 131.372,Z 275.492,A -85,B 0,C 180,E1 -25120.013,E2 -25120.013} C_VEL
LIN {X 0,Y 134.253,Z 268.18,A -85,B 0,C 180,E1 -25124.398,E2 -25124.398} C_VEL
LIN {X 0,Y 137.603,Z 259.138,A -85,B 0,C 180,E1 -25128.616,E2 -25128.616} C_VEL
LIN {X 0,Y 141.027,Z 249.723,A -85,B 0,C 180,E1 -25131.948,E2 -25131.948} C_VEL
LIN {X 0,Y 144.581,Z 239.245,A -85,B 0,C 180,E1 -25134.788,E2 -25134.788} C_VEL
LIN {X 0,Y 147.788,Z 227.641,A -85,B 0,C 180,E1 -25137.24,E2 -25137.24} C_VEL
LIN {X 0,Y 150.439,Z 215.317,A -85,B 0,C 180,E1 -25139.184,E2 -25139.184} C_VEL
LIN {X 0,Y 152.51,Z 202.207,A -85,B 0,C 180,E1 -25140.672,E2 -25140.672} C_VEL
LIN {X 0,Y 153.757,Z 190.372,A -85,B 0,C 180,E1 -25141.566,E2 -25141.566} C_VEL
LIN {X 0,Y 156.625,Z 142.873,A -85,B 0,C 180,E1 -25143.562,E2 -25143.562} C_VEL
LIN {X 0,Y 150.957,Z 130.812,A -85,B 0,C 180,E1 -25146.107,E2 -25146.107} C_VEL
LIN {X 0,Y 144.949,Z 120.126,A -85,B 0,C 180,E1 -25149.007,E2 -25149.007} C_VEL
LIN {X 0,Y 140.071,Z 112.696,A -85,B 0,C 180,E1 -25151.571,E2 -25151.571} C_VEL
LIN {X 0,Y 137.903,Z 109.552,A -85,B 0,C 180,E1 -25152.799,E2 -25152.799} C_VEL
LIN {X 0,Y 135.5,Z 106.086,A -85,B 0,C 180,E1 -25154.241,E2 -25154.241} C_VEL
LIN {X 0,Y 133.122,Z 103.048,A -85,B 0,C 180,E1 -25155.731,E2 -25155.731} C_VEL
LIN {X 0,Y 132.464,Z 101.709,A -85,B 0,C 180,E1 -25156.205,E2 -25156.205} C_VEL
LIN {X 0,Y 130.185,Z 99.621,A -85,B 0,C 180,E1 -25157.692,E2 -25157.692} C_VEL
LIN {X 0,Y 129.098,Z 97.276,A -85,B 0,C 180,E1 -25158.565,E2 -25158.565} C_VEL
LIN {X 0,Y 128.941,Z 96.415,A -85,B 0,C 180,E1 -25158.763,E2 -25158.763} C_VEL
LIN {X 0,Y 128.982,Z 96.407,A -85,B 0,C 180,E1 -25164.819,E2 -25164.819} C_VEL
LIN {X 0,Y 129.053,Z 96.402,A -85,B 0,C 180,E1 -25170.652,E2 -25170.652} C_VEL
LIN {X 0,Y 129.11,Z 96.403,A -85,B 0,C 180,E1 -25177.728,E2 -25177.728} C_VEL
LIN {X 0,Y 129.185,Z 96.35,A -85,B 0,C 180,E1 -25184.216,E2 -25184.216} C_VEL
LIN {X 0,Y 129.378,Z 96.363,A -85,B 0,C 180,E1 -25187.904,E2 -25187.904} C_VEL
LIN {X 0,Y 129.477,Z 96.354,A -85,B 0,C 180,E1 -25190.629,E2 -25190.629} C_VEL
LIN {X 0,Y 130.09,Z 96.275,A -85,B 0,C 180,E1 -25200,E2 -25200} C_VEL
LIN {X 0,Y 129.475,Z 96.348,A -85,B 0,C 180,E1 -25209.372,E2 -25209.372} C_VEL
LIN {X 0,Y 129.346,Z 96.373,A -85,B 0,C 180,E1 -25212.553,E2 -25212.553} C_VEL
LIN {X 0,Y 129.151,Z 96.395,A -85,B 0,C 180,E1 -25219.057,E2 -25219.057} C_VEL
LIN {X 0,Y 129.11,Z 96.405,A -85,B 0,C 180,E1 -25222.399,E2 -25222.399} C_VEL
LIN {X 0,Y 129.019,Z 96.418,A -85,B 0,C 180,E1 -25229.358,E2 -25229.358} C_VEL
LIN {X 0,Y 129.044,Z 96.584,A -85,B 0,C 180,E1 -25230.59,E2 -25230.59} C_VEL
LIN {X 0,Y 129.939,Z 99.145,A -85,B 0,C 180,E1 -25231.372,E2 -25231.372} C_VEL
LIN {X 0,Y 131.899,Z 101.326,A -85,B 0,C 180,E1 -25232.702,E2 -25232.702} C_VEL
LIN {X 0,Y 132.73,Z 102.069,A -85,B 0,C 180,E1 -25233.226,E2 -25233.226} C_VEL
LIN {X 0,Y 134.843,Z 105.415,A -85,B 0,C 180,E1 -25234.625,E2 -25234.625} C_VEL
LIN {X 0,Y 136.384,Z 107.249,A -85,B 0,C 180,E1 -25235.545,E2 -25235.545} C_VEL
LIN {X 0,Y 139.834,Z 112.304,A -85,B 0,C 180,E1 -25237.547,E2 -25237.547} C_VEL
LIN {X 0,Y 144.087,Z 120.385,A -85,B 0,C 180,E1 -25239.92,E2 -25239.92} C_VEL
LIN {X 0,Y 148.98,Z 130.988,A -85,B 0,C 180,E1 -25242.469,E2 -25242.469} C_VEL
LIN {X 0,Y 153.51,Z 143.111,A -85,B 0,C 180,E1 -25244.741,E2 -25244.741} C_VEL
LIN {X 0,Y 154.165,Z 145.729,A -85,B 0,C 180,E1 -25245.104,E2 -25245.104} C_VEL
LIN {X 0,Y 155.333,Z 165.556,A -85,B 0,C 180,E1 -25246.626,E2 -25246.626} C_VEL
LIN {X 0,Y 152.883,Z 204.776,A -85,B 0,C 180,E1 -25248.308,E2 -25248.308} C_VEL
LIN {X 0,Y 151.099,Z 218.529,A -85,B 0,C 180,E1 -25249.369,E2 -25249.369} C_VEL
LIN {X 0,Y 148.691,Z 230.851,A -85,B 0,C 180,E1 -25250.788,E2 -25250.788} C_VEL
LIN {X 0,Y 145.397,Z 243.492,A -85,B 0,C 180,E1 -25252.828,E2 -25252.828} C_VEL
LIN {X 0,Y 142.021,Z 254.784,A -85,B 0,C 180,E1 -25255.313,E2 -25255.313} C_VEL
LIN {X 0,Y 139.314,Z 262.833,A -85,B 0,C 180,E1 -25257.588,E2 -25257.588} C_VEL
LIN {X 0,Y 136.239,Z 271.548,A -85,B 0,C 180,E1 -25260.655,E2 -25260.655} C_VEL
LIN {X 0,Y 133.062,Z 279.431,A -85,B 0,C 180,E1 -25264.108,E2 -25264.108} C_VEL
LIN {X 0,Y 130.808,Z 286.205,A -85,B 0,C 180,E1 -25267.908,E2 -25267.908} C_VEL
LIN {X 0,Y 128.678,Z 292.742,A -85,B 0,C 180,E1 -25272.518,E2 -25272.518} C_VEL
LIN {X 0,Y 127.293,Z 297.914,A -85,B 0,C 180,E1 -25277.241,E2 -25277.241} C_VEL
LIN {X 0,Y 126.685,Z 301.918,A -85,B 0,C 180,E1 -25282.028,E2 -25282.028} C_VEL
LIN {X 0,Y 126.7,Z 304.856,A -85,B 0,C 180,E1 -25286.82,E2 -25286.82} C_VEL
LIN {X 0,Y 126.9,Z 306.23,A -85,B 0,C 180,E1 -25290,E2 -25290} C_VEL
LIN {X 0,Y 126.742,Z 307.237,A -85,B 0,C 180,E1 -25293.5,E2 -25293.5} C_VEL
LIN {X 0,Y 126.773,Z 307.824,A -85,B 0,C 180,E1 -25299.573,E2 -25299.573} C_VEL
LIN {X 0,Y 128.256,Z 306.876,A -85,B 0,C 180,E1 -25305.901,E2 -25305.901} C_VEL
LIN {X 0,Y 131.326,Z 304.406,A -85,B 0,C 180,E1 -25312,E2 -25312} C_VEL
LIN {X 0,Y 134.735,Z 301.332,A -85,B 0,C 180,E1 -25316.468,E2 -25316.468} C_VEL
LIN {X 0,Y 136.122,Z 299.401,A -85,B 0,C 180,E1 -25318.748,E2 -25318.748} C_VEL
LIN {X 0,Y 137.107,Z 295.781,A -85,B 0,C 180,E1 -25322.609,E2 -25322.609} C_VEL
LIN {X 0,Y 138.602,Z 291.659,A -85,B 0,C 180,E1 -25326.297,E2 -25326.297} C_VEL
LIN {X 0,Y 140.701,Z 288.748,A -85,B 0,C 180,E1 -25328.223,E2 -25328.223} C_VEL
LIN {X 0,Y 147.26,Z 281.003,A -85,B 0,C 180,E1 -25331.925,E2 -25331.925} C_VEL
LIN {X 0,Y 153.949,Z 272.014,A -85,B 0,C 180,E1 -25335.04,E2 -25335.04} C_VEL
LIN {X 0,Y 159.808,Z 262.79,A -85,B 0,C 180,E1 -25337.445,E2 -25337.445} C_VEL
LIN {X 0,Y 165.483,Z 252.54,A -85,B 0,C 180,E1 -25339.389,E2 -25339.389} C_VEL
LIN {X 0,Y 169.964,Z 242.785,A -85,B 0,C 180,E1 -25340.833,E2 -25340.833} C_VEL
LIN {X 0,Y 174.592,Z 230.438,A -85,B 0,C 180,E1 -25342.184,E2 -25342.184} C_VEL
LIN {X 0,Y 177.871,Z 219.002,A -85,B 0,C 180,E1 -25343.094,E2 -25343.094} C_VEL
LIN {X 0,Y 180.476,Z 206.376,A -85,B 0,C 180,E1 -25343.762,E2 -25343.762} C_VEL
LIN {X 0,Y 182.198,Z 190.492,A -85,B 0,C 180,E1 -25344.33,E2 -25344.33} C_VEL
LIN {X 0,Y 182.798,Z 182.567,A -85,B 0,C 180,E1 -25344.612,E2 -25344.612} C_VEL
LIN {X 0,Y 179.616,Z 173.585,A -85,B 0,C 180,E1 -25347.071,E2 -25347.071} C_VEL
LIN {X 0,Y 176.216,Z 165.217,A -85,B 0,C 180,E1 -25349.932,E2 -25349.932} C_VEL
LIN {X 0,Y 173.162,Z 158.316,A -85,B 0,C 180,E1 -25352.829,E2 -25352.829} C_VEL
LIN {X 0,Y 170.596,Z 153.083,A -85,B 0,C 180,E1 -25355.592,E2 -25355.592} C_VEL
LIN {X 0,Y 168.769,Z 149.348,A -85,B 0,C 180,E1 -25357.869,E2 -25357.869} C_VEL
LIN {X 0,Y 166.299,Z 144.512,A -85,B 0,C 180,E1 -25361.607,E2 -25361.607} C_VEL
LIN {X 0,Y 164.18,Z 141.503,A -85,B 0,C 180,E1 -25365.751,E2 -25365.751} C_VEL
LIN {X 0,Y 163.562,Z 139.914,A -85,B 0,C 180,E1 -25367.593,E2 -25367.593} C_VEL
LIN {X 0,Y 162.34,Z 139.005,A -85,B 0,C 180,E1 -25372.537,E2 -25372.537} C_VEL
LIN {X 0,Y 162.444,Z 138.798,A -85,B 0,C 180,E1 -25378.76,E2 -25378.76} C_VEL
LIN {X 0,Y 163.829,Z 140.059,A -85,B 0,C 180,E1 -25383.882,E2 -25383.882} C_VEL
LIN {X 0,Y 165.595,Z 143.56,A -85,B 0,C 180,E1 -25387.966,E2 -25387.966} C_VEL
LIN {X 0,Y 166.728,Z 144.971,A -85,B 0,C 180,E1 -25389.836,E2 -25389.836} C_VEL
LIN {X 0,Y 169.526,Z 149.46,A -85,B 0,C 180,E1 -25393.714,E2 -25393.714} C_VEL
LIN {X 0,Y 172.402,Z 154.074,A -85,B 0,C 180,E1 -25396.885,E2 -25396.885} C_VEL
LIN {X 0,Y 175.235,Z 158.688,A -85,B 0,C 180,E1 -25399.55,E2 -25399.55} C_VEL
LIN {X 0,Y 179.437,Z 166.1,A -85,B 0,C 180,E1 -25402.982,E2 -25402.982} C_VEL
LIN {X 0,Y 183.493,Z 174.174,A -85,B 0,C 180,E1 -25405.901,E2 -25405.901} C_VEL
LIN {X 0,Y 181.54,Z 194.073,A -85,B 0,C 180,E1 -25406.571,E2 -25406.571} C_VEL
LIN {X 0,Y 179.285,Z 206.977,A -85,B 0,C 180,E1 -25407.341,E2 -25407.341} C_VEL
LIN {X 0,Y 176.426,Z 218.354,A -85,B 0,C 180,E1 -25408.341,E2 -25408.341} C_VEL
LIN {X 0,Y 172.328,Z 230.411,A -85,B 0,C 180,E1 -25409.762,E2 -25409.762} C_VEL
LIN {X 0,Y 167.133,Z 242.334,A -85,B 0,C 180,E1 -25411.622,E2 -25411.622} C_VEL
LIN {X 0,Y 161.663,Z 252.574,A -85,B 0,C 180,E1 -25413.755,E2 -25413.755} C_VEL
LIN {X 0,Y 155.439,Z 262.592,A -85,B 0,C 180,E1 -25416.626,E2 -25416.626} C_VEL
LIN {X 0,Y 149.938,Z 269.99,A -85,B 0,C 180,E1 -25419.34,E2 -25419.34} C_VEL
LIN {X 0,Y 143.883,Z 277.225,A -85,B 0,C 180,E1 -25422.888,E2 -25422.888} C_VEL
LIN {X 0,Y 138.405,Z 282.932,A -85,B 0,C 180,E1 -25426.724,E2 -25426.724} C_VEL
LIN {X 0,Y 133.468,Z 287.384,A -85,B 0,C 180,E1 -25430.811,E2 -25430.811} C_VEL
LIN {X 0,Y 130.379,Z 289.893,A -85,B 0,C 180,E1 -25433.956,E2 -25433.956} C_VEL
LIN {X 0,Y 128.054,Z 291.603,A -85,B 0,C 180,E1 -25436.713,E2 -25436.713} C_VEL
LIN {X 0,Y 125.814,Z 293.029,A -85,B 0,C 180,E1 -25439.819,E2 -25439.819} C_VEL
LIN {X 0,Y 122.404,Z 294.601,A -85,B 0,C 180,E1 -25446.302,E2 -25446.302} C_VEL
LIN {X 0,Y 121.172,Z 294.799,A -85,B 0,C 180,E1 -25449.635,E2 -25449.635} C_VEL
LIN {X 0,Y 120.28,Z 294.558,A -85,B 0,C 180,E1 -25453.013,E2 -25453.013} C_VEL
LIN {X 0,Y 119.513,Z 292.883,A -85,B 0,C 180,E1 -25459.839,E2 -25459.839} C_VEL
LIN {X 0,Y 119.923,Z 290.484,A -85,B 0,C 180,E1 -25465.046,E2 -25465.046} C_VEL
LIN {X 0,Y 120.604,Z 287.233,A -85,B 0,C 180,E1 -25470,E2 -25470} C_VEL
LIN {X 0,Y 122.008,Z 282.871,A -85,B 0,C 180,E1 -25474.957,E2 -25474.957} C_VEL
LIN {X 0,Y 123.987,Z 277.338,A -85,B 0,C 180,E1 -25479.791,E2 -25479.791} C_VEL
LIN {X 0,Y 126.825,Z 270.423,A -85,B 0,C 180,E1 -25484.44,E2 -25484.44} C_VEL
LIN {X 0,Y 130.285,Z 261.764,A -85,B 0,C 180,E1 -25488.885,E2 -25488.885} C_VEL
LIN {X 0,Y 133.701,Z 252.893,A -85,B 0,C 180,E1 -25492.402,E2 -25492.402} C_VEL
LIN {X 0,Y 137.277,Z 243.118,A -85,B 0,C 180,E1 -25495.39,E2 -25495.39} C_VEL
LIN {X 0,Y 140.702,Z 232.372,A -85,B 0,C 180,E1 -25497.923,E2 -25497.923} C_VEL
LIN {X 0,Y 143.709,Z 220.369,A -85,B 0,C 180,E1 -25500.084,E2 -25500.084} C_VEL
LIN {X 0,Y 146.073,Z 207.891,A -85,B 0,C 180,E1 -25501.752,E2 -25501.752} C_VEL
LIN {X 0,Y 147.728,Z 195.249,A -85,B 0,C 180,E1 -25502.918,E2 -25502.918} C_VEL
LIN {X 0,Y 148.946,Z 179.556,A -85,B 0,C 180,E1 -25503.733,E2 -25503.733} C_VEL
LIN {X 0,Y 151.027,Z 145.014,A -85,B 0,C 180,E1 -25505.195,E2 -25505.195} C_VEL
LIN {X 0,Y 145.555,Z 133.331,A -85,B 0,C 180,E1 -25507.877,E2 -25507.877} C_VEL
LIN {X 0,Y 139.466,Z 122.571,A -85,B 0,C 180,E1 -25511.104,E2 -25511.104} C_VEL
LIN {X 0,Y 134.247,Z 114.739,A -85,B 0,C 180,E1 -25514.167,E2 -25514.167} C_VEL
LIN {X 0,Y 132.114,Z 111.644,A -85,B 0,C 180,E1 -25515.541,E2 -25515.541} C_VEL
LIN {X 0,Y 129.592,Z 108.101,A -85,B 0,C 180,E1 -25517.268,E2 -25517.268} C_VEL
LIN {X 0,Y 126.604,Z 104.429,A -85,B 0,C 180,E1 -25519.453,E2 -25519.453} C_VEL
LIN {X 0,Y 125.612,Z 102.699,A -85,B 0,C 180,E1 -25520.281,E2 -25520.281} C_VEL
LIN {X 0,Y 123.188,Z 100.642,A -85,B 0,C 180,E1 -25522.209,E2 -25522.209} C_VEL
LIN {X 0,Y 122.087,Z 98.231,A -85,B 0,C 180,E1 -25523.313,E2 -25523.313} C_VEL
LIN {X 0,Y 121.913,Z 97.289,A -85,B 0,C 180,E1 -25523.677,E2 -25523.677} C_VEL
LIN {X 0,Y 121.943,Z 97.284,A -85,B 0,C 180,E1 -25529.827,E2 -25529.827} C_VEL
LIN {X 0,Y 121.985,Z 97.283,A -85,B 0,C 180,E1 -25536.216,E2 -25536.216} C_VEL
LIN {X 0,Y 122.036,Z 97.272,A -85,B 0,C 180,E1 -25539.786,E2 -25539.786} C_VEL
LIN {X 0,Y 122.24,Z 97.234,A -85,B 0,C 180,E1 -25546.705,E2 -25546.705} C_VEL
LIN {X 0,Y 122.409,Z 97.236,A -85,B 0,C 180,E1 -25550.082,E2 -25550.082} C_VEL
LIN {X 0,Y 122.597,Z 97.171,A -85,B 0,C 180,E1 -25556.714,E2 -25556.714} C_VEL
LIN {X 0,Y 123.044,Z 97.152,A -85,B 0,C 180,E1 -25560,E2 -25560} C_VEL
LIN {X 0,Y 122.423,Z 97.235,A -85,B 0,C 180,E1 -25566.593,E2 -25566.593} C_VEL
LIN {X 0,Y 122.325,Z 97.247,A -85,B 0,C 180,E1 -25572.386,E2 -25572.386} C_VEL
LIN {X 0,Y 122.106,Z 97.27,A -85,B 0,C 180,E1 -25576.726,E2 -25576.726} C_VEL
LIN {X 0,Y 122.029,Z 97.288,A -85,B 0,C 180,E1 -25582.854,E2 -25582.854} C_VEL
LIN {X 0,Y 121.984,Z 97.287,A -85,B 0,C 180,E1 -25585.716,E2 -25585.716} C_VEL
LIN {X 0,Y 122.807,Z 99.894,A -85,B 0,C 180,E1 -25586.673,E2 -25586.673} C_VEL
LIN {X 0,Y 124.698,Z 102.054,A -85,B 0,C 180,E1 -25588.273,E2 -25588.273} C_VEL
LIN {X 0,Y 126.053,Z 103.15,A -85,B 0,C 180,E1 -25589.307,E2 -25589.307} C_VEL
LIN {X 0,Y 127.888,Z 106.218,A -85,B 0,C 180,E1 -25590.782,E2 -25590.782} C_VEL
LIN {X 0,Y 129.768,Z 108.288,A -85,B 0,C 180,E1 -25592.102,E2 -25592.102} C_VEL
LIN {X 0,Y 132.381,Z 111.913,A -85,B 0,C 180,E1 -25593.879,E2 -25593.879} C_VEL
LIN {X 0,Y 136.489,Z 118.115,A -85,B 0,C 180,E1 -25596.453,E2 -25596.453} C_VEL
LIN {X 0,Y 140.967,Z 127.137,A -85,B 0,C 180,E1 -25599.123,E2 -25599.123} C_VEL
LIN {X 0,Y 145.307,Z 137.417,A -85,B 0,C 180,E1 -25601.555,E2 -25601.555} C_VEL
LIN {X 0,Y 148.793,Z 147.432,A -85,B 0,C 180,E1 -25603.456,E2 -25603.456} C_VEL
LIN {X 0,Y 149.753,Z 166.71,A -85,B 0,C 180,E1 -25604.982,E2 -25604.982} C_VEL
LIN {X 0,Y 147.327,Z 204.186,A -85,B 0,C 180,E1 -25606.634,E2 -25606.634} C_VEL
LIN {X 0,Y 145.463,Z 217.697,A -85,B 0,C 180,E1 -25607.67,E2 -25607.67} C_VEL
LIN {X 0,Y 142.999,Z 230.185,A -85,B 0,C 180,E1 -25609.135,E2 -25609.135} C_VEL
LIN {X 0,Y 139.798,Z 242.092,A -85,B 0,C 180,E1 -25611.067,E2 -25611.067} C_VEL
LIN {X 0,Y 136.227,Z 253.569,A -85,B 0,C 180,E1 -25613.609,E2 -25613.609} C_VEL
LIN {X 0,Y 133.28,Z 261.747,A -85,B 0,C 180,E1 -25615.925,E2 -25615.925} C_VEL
LIN {X 0,Y 130.023,Z 270.582,A -85,B 0,C 180,E1 -25619.103,E2 -25619.103} C_VEL
LIN {X 0,Y 126.978,Z 277.986,A -85,B 0,C 180,E1 -25622.419,E2 -25622.419} C_VEL
LIN {X 0,Y 124.202,Z 285.421,A -85,B 0,C 180,E1 -25626.665,E2 -25626.665} C_VEL
LIN {X 0,Y 121.892,Z 292.045,A -85,B 0,C 180,E1 -25631.511,E2 -25631.511} C_VEL
LIN {X 0,Y 120.33,Z 297.292,A -85,B 0,C 180,E1 -25636.489,E2 -25636.489} C_VEL
LIN {X 0,Y 119.646,Z 301.357,A -85,B 0,C 180,E1 -25641.555,E2 -25641.555} C_VEL
LIN {X 0,Y 119.617,Z 304.615,A -85,B 0,C 180,E1 -25647.225,E2 -25647.225} C_VEL
LIN {X 0,Y 119.802,Z 305.757,A -85,B 0,C 180,E1 -25650,E2 -25650} C_VEL
LIN {X 0,Y 119.684,Z 306.714,A -85,B 0,C 180,E1 -25653.366,E2 -25653.366} C_VEL
LIN {X 0,Y 119.759,Z 307.433,A -85,B 0,C 180,E1 -25660.14,E2 -25660.14} C_VEL
LIN {X 0,Y 120.408,Z 307.194,A -85,B 0,C 180,E1 -25663.501,E2 -25663.501} C_VEL
LIN {X 0,Y 122.836,Z 305.536,A -85,B 0,C 180,E1 -25670.077,E2 -25670.077} C_VEL
LIN {X 0,Y 124.755,Z 304.137,A -85,B 0,C 180,E1 -25673.225,E2 -25673.225} C_VEL
LIN {X 0,Y 128.288,Z 301.225,A -85,B 0,C 180,E1 -25677.753,E2 -25677.753} C_VEL
LIN {X 0,Y 132.479,Z 297.307,A -85,B 0,C 180,E1 -25682.039,E2 -25682.039} C_VEL
LIN {X 0,Y 137.393,Z 292.291,A -85,B 0,C 180,E1 -25686.033,E2 -25686.033} C_VEL
LIN {X 0,Y 140.701,Z 288.748,A -85,B 0,C 180,E1 -25688.223,E2 -25688.223} C_VEL
LIN {X 0,Y 142.963,Z 285.661,A -85,B 0,C 180,E1 -25690.045,E2 -25690.045} C_VEL
LIN {X 0,Y 145.444,Z 280.292,A -85,B 0,C 180,E1 -25693.21,E2 -25693.21} C_VEL
LIN {X 0,Y 148.02,Z 274.322,A -85,B 0,C 180,E1 -25696.13,E2 -25696.13} C_VEL
LIN {X 0,Y 150.335,Z 270.296,A -85,B 0,C 180,E1 -25697.534,E2 -25697.534} C_VEL
LIN {X 0,Y 157.011,Z 259.911,A -85,B 0,C 180,E1 -25700.044,E2 -25700.044} C_VEL
LIN {X 0,Y 162.222,Z 250.435,A -85,B 0,C 180,E1 -25701.743,E2 -25701.743} C_VEL
LIN {X 0,Y 167.611,Z 238.68,A -85,B 0,C 180,E1 -25703.314,E2 -25703.314} C_VEL
LIN {X 0,Y 172.073,Z 226.112,A -85,B 0,C 180,E1 -25704.519,E2 -25704.519} C_VEL
LIN {X 0,Y 175.546,Z 212.865,A -85,B 0,C 180,E1 -25705.408,E2 -25705.408} C_VEL
LIN {X 0,Y 177.575,Z 200.851,A -85,B 0,C 180,E1 -25705.953,E2 -25705.953} C_VEL
LIN {X 0,Y 178.986,Z 185.24,A -85,B 0,C 180,E1 -25706.484,E2 -25706.484} C_VEL
LIN {X 0,Y 176.283,Z 177.42,A -85,B 0,C 180,E1 -25708.783,E2 -25708.783} C_VEL
LIN {X 0,Y 173.362,Z 169.85,A -85,B 0,C 180,E1 -25711.496,E2 -25711.496} C_VEL
LIN {X 0,Y 170.552,Z 163.256,A -85,B 0,C 180,E1 -25714.435,E2 -25714.435} C_VEL
LIN {X 0,Y 168.477,Z 158.723,A -85,B 0,C 180,E1 -25716.915,E2 -25716.915} C_VEL
LIN {X 0,Y 167.04,Z 155.585,A -85,B 0,C 180,E1 -25718.884,E2 -25718.884} C_VEL
LIN {X 0,Y 165.036,Z 151.306,A -85,B 0,C 180,E1 -25722.179,E2 -25722.179} C_VEL
LIN {X 0,Y 163,Z 148.186,A -85,B 0,C 180,E1 -25726.48,E2 -25726.48} C_VEL
LIN {X 0,Y 162.491,Z 146.863,A -85,B 0,C 180,E1 -25728.131,E2 -25728.131} C_VEL
LIN {X 0,Y 161.473,Z 146.06,A -85,B 0,C 180,E1 -25732.497,E2 -25732.497} C_VEL
LIN {X 0,Y 161.41,Z 145.738,A -85,B 0,C 180,E1 -25737.504,E2 -25737.504} C_VEL
LIN {X 0,Y 162.666,Z 146.797,A -85,B 0,C 180,E1 -25743.096,E2 -25743.096} C_VEL
LIN {X 0,Y 164.708,Z 150.783,A -85,B 0,C 180,E1 -25748.009,E2 -25748.009} C_VEL
LIN {X 0,Y 165.462,Z 151.914,A -85,B 0,C 180,E1 -25749.319,E2 -25749.319} C_VEL
LIN {X 0,Y 167.98,Z 156.126,A -85,B 0,C 180,E1 -25753.015,E2 -25753.015} C_VEL
LIN {X 0,Y 170.592,Z 160.507,A -85,B 0,C 180,E1 -25756.069,E2 -25756.069} C_VEL
LIN {X 0,Y 173.76,Z 165.879,A -85,B 0,C 180,E1 -25759.185,E2 -25759.185} C_VEL
LIN {X 0,Y 178.093,Z 174.268,A -85,B 0,C 180,E1 -25762.858,E2 -25762.858} C_VEL
LIN {X 0,Y 179.626,Z 177.454,A -85,B 0,C 180,E1 -25764.034,E2 -25764.034} C_VEL
LIN {X 0,Y 177.845,Z 194.82,A -85,B 0,C 180,E1 -25764.645,E2 -25764.645} C_VEL
LIN {X 0,Y 175.416,Z 208.09,A -85,B 0,C 180,E1 -25765.448,E2 -25765.448} C_VEL
LIN {X 0,Y 171.944,Z 220.807,A -85,B 0,C 180,E1 -25766.601,E2 -25766.601} C_VEL
LIN {X 0,Y 167.345,Z 233.284,A -85,B 0,C 180,E1 -25768.122,E2 -25768.122} C_VEL
LIN {X 0,Y 162.161,Z 244.287,A -85,B 0,C 180,E1 -25769.911,E2 -25769.911} C_VEL
LIN {X 0,Y 157.126,Z 253.215,A -85,B 0,C 180,E1 -25771.806,E2 -25771.806} C_VEL
LIN {X 0,Y 151.222,Z 262.367,A -85,B 0,C 180,E1 -25774.419,E2 -25774.419} C_VEL
LIN {X 0,Y 145.426,Z 269.866,A -85,B 0,C 180,E1 -25777.118,E2 -25777.118} C_VEL
LIN {X 0,Y 139.036,Z 277.196,A -85,B 0,C 180,E1 -25780.692,E2 -25780.692} C_VEL
LIN {X 0,Y 133.201,Z 283.009,A -85,B 0,C 180,E1 -25784.578,E2 -25784.578} C_VEL
LIN {X 0,Y 127.907,Z 287.536,A -85,B 0,C 180,E1 -25788.749,E2 -25788.749} C_VEL
LIN {X 0,Y 124.142,Z 290.385,A -85,B 0,C 180,E1 -25792.426,E2 -25792.426} C_VEL
LIN {X 0,Y 119.577,Z 293.31,A -85,B 0,C 180,E1 -25798.065,E2 -25798.065} C_VEL
LIN {X 0,Y 115.791,Z 294.947,A -85,B 0,C 180,E1 -25804.858,E2 -25804.858} C_VEL
LIN {X 0,Y 114.417,Z 295.176,A -85,B 0,C 180,E1 -25808.374,E2 -25808.374} C_VEL
LIN {X 0,Y 113.382,Z 294.996,A -85,B 0,C 180,E1 -25811.945,E2 -25811.945} C_VEL
LIN {X 0,Y 112.435,Z 293.381,A -85,B 0,C 180,E1 -25819.192,E2 -25819.192} C_VEL
LIN {X 0,Y 112.847,Z 290.818,A -85,B 0,C 180,E1 -25825.175,E2 -25825.175} C_VEL
LIN {X 0,Y 113.507,Z 287.854,A -85,B 0,C 180,E1 -25830,E2 -25830} C_VEL
LIN {X 0,Y 114.941,Z 283.562,A -85,B 0,C 180,E1 -25835.263,E2 -25835.263} C_VEL
LIN {X 0,Y 117.431,Z 277.097,A -85,B 0,C 180,E1 -25841.216,E2 -25841.216} C_VEL
LIN {X 0,Y 120.563,Z 269.98,A -85,B 0,C 180,E1 -25846.075,E2 -25846.075} C_VEL
LIN {X 0,Y 124.292,Z 261.142,A -85,B 0,C 180,E1 -25850.696,E2 -25850.696} C_VEL
LIN {X 0,Y 127.988,Z 252.067,A -85,B 0,C 180,E1 -25854.321,E2 -25854.321} C_VEL
LIN {X 0,Y 131.799,Z 241.992,A -85,B 0,C 180,E1 -25857.382,E2 -25857.382} C_VEL
LIN {X 0,Y 135.408,Z 230.806,A -85,B 0,C 180,E1 -25859.971,E2 -25859.971} C_VEL
LIN {X 0,Y 138.582,Z 218.31,A -85,B 0,C 180,E1 -25862.175,E2 -25862.175} C_VEL
LIN {X 0,Y 140.904,Z 205.702,A -85,B 0,C 180,E1 -25863.78,E2 -25863.78} C_VEL
LIN {X 0,Y 142.587,Z 192.344,A -85,B 0,C 180,E1 -25864.907,E2 -25864.907} C_VEL
LIN {X 0,Y 145.247,Z 154.476,A -85,B 0,C 180,E1 -25866.582,E2 -25866.582} C_VEL
LIN {X 0,Y 145.647,Z 147.38,A -85,B 0,C 180,E1 -25866.906,E2 -25866.906} C_VEL
LIN {X 0,Y 140.467,Z 136.264,A -85,B 0,C 180,E1 -25869.679,E2 -25869.679} C_VEL
LIN {X 0,Y 135.424,Z 127.286,A -85,B 0,C 180,E1 -25872.585,E2 -25872.585} C_VEL
LIN {X 0,Y 130.906,Z 120.269,A -85,B 0,C 180,E1 -25875.452,E2 -25875.452} C_VEL
LIN {X 0,Y 128.47,Z 116.764,A -85,B 0,C 180,E1 -25877.136,E2 -25877.136} C_VEL
LIN {X 0,Y 125.795,Z 113.02,A -85,B 0,C 180,E1 -25879.137,E2 -25879.137} C_VEL
LIN {X 0,Y 123.213,Z 109.269,A -85,B 0,C 180,E1 -25881.271,E2 -25881.271} C_VEL
LIN {X 0,Y 120.35,Z 106.248,A -85,B 0,C 180,E1 -25883.776,E2 -25883.776} C_VEL
LIN {X 0,Y 119.076,Z 103.794,A -85,B 0,C 180,E1 -25885.127,E2 -25885.127} C_VEL
LIN {X 0,Y 116.508,Z 101.952,A -85,B 0,C 180,E1 -25887.711,E2 -25887.711} C_VEL
LIN {X 0,Y 115.171,Z 99.444,A -85,B 0,C 180,E1 -25889.426,E2 -25889.426} C_VEL
LIN {X 0,Y 114.91,Z 98.16,A -85,B 0,C 180,E1 -25889.985,E2 -25889.985} C_VEL
LIN {X 0,Y 114.949,Z 98.16,A -85,B 0,C 180,E1 -25896.508,E2 -25896.508} C_VEL
LIN {X 0,Y 115.003,Z 98.117,A -85,B 0,C 180,E1 -25902.209,E2 -25902.209} C_VEL
LIN {X 0,Y 115.257,Z 98.111,A -85,B 0,C 180,E1 -25907.327,E2 -25907.327} C_VEL
LIN {X 0,Y 115.366,Z 98.08,A -85,B 0,C 180,E1 -25913.002,E2 -25913.002} C_VEL
LIN {X 0,Y 115.995,Z 98.029,A -85,B 0,C 180,E1 -25920,E2 -25920} C_VEL
LIN {X 0,Y 115.364,Z 98.115,A -85,B 0,C 180,E1 -25926.999,E2 -25926.999} C_VEL
LIN {X 0,Y 115.257,Z 98.128,A -85,B 0,C 180,E1 -25932.673,E2 -25932.673} C_VEL
LIN {X 0,Y 114.978,Z 98.158,A -85,B 0,C 180,E1 -25939.413,E2 -25939.413} C_VEL
LIN {X 0,Y 115.873,Z 100.814,A -85,B 0,C 180,E1 -25940.759,E2 -25940.759} C_VEL
LIN {X 0,Y 117.743,Z 102.948,A -85,B 0,C 180,E1 -25942.843,E2 -25942.843} C_VEL
LIN {X 0,Y 119.312,Z 103.99,A -85,B 0,C 180,E1 -25944.352,E2 -25944.352} C_VEL
LIN {X 0,Y 121.079,Z 107.145,A -85,B 0,C 180,E1 -25946.154,E2 -25946.154} C_VEL
LIN {X 0,Y 123.302,Z 109.351,A -85,B 0,C 180,E1 -25948.05,E2 -25948.05} C_VEL
LIN {X 0,Y 125.714,Z 112.889,A -85,B 0,C 180,E1 -25950.045,E2 -25950.045} C_VEL
LIN {X 0,Y 127.002,Z 114.549,A -85,B 0,C 180,E1 -25951.02,E2 -25951.02} C_VEL
LIN {X 0,Y 130.363,Z 119.452,A -85,B 0,C 180,E1 -25953.43,E2 -25953.43} C_VEL
LIN {X 0,Y 132.838,Z 123.276,A -85,B 0,C 180,E1 -25955.07,E2 -25955.07} C_VEL
LIN {X 0,Y 137.238,Z 132.676,A -85,B 0,C 180,E1 -25957.918,E2 -25957.918} C_VEL
LIN {X 0,Y 141.336,Z 142.841,A -85,B 0,C 180,E1 -25960.39,E2 -25960.39} C_VEL
LIN {X 0,Y 143.648,Z 149.94,A -85,B 0,C 180,E1 -25961.777,E2 -25961.777} C_VEL
